# B&R Automation Studio project OpcUaSample410_BrbLibUa103
Automation Studio 4.10.4.38 SP

## Configuration ArSim

CPU PC_any, AutomationRuntime H4.91, Build 6.3.0, Vc V4.16.2

CPU X20CP0483, AutomationRuntime H4.91, Build 6.3.0, Vc V4.16.2

### Task classes (Cpu.sw)
```
Cyclic#1 (cycle 10000 us):
  ClientC <- Tasks.Clients.ClientC.ClientC.prg
  ClientST <- Tasks.Clients.ClientST.ClientST.prg
  SrvMethC <- Tasks.ServerMethods.SrvMethC.SrvMethC.prg
  SrvMethST <- Tasks.ServerMethods.SrvMethST.SrvMethST.prg
  SrvEvntC <- Tasks.ServerEvents.SrvEvntC.SrvEvntC.prg
  SrvEvntST <- Tasks.ServerEvents.SrvEvntST.SrvEvntST.prg [disabled]
  BrbUaCltC <- Tasks.BrbUa.BrbUaClient.BrbUaCltC.BrbUaCltC.prg
  BrbUaCltST <- Tasks.BrbUa.BrbUaClient.BrbUaCltST.BrbUaCltST.prg
  BrbUaSrvC <- Tasks.BrbUa.BrbUaServer.BrbUaSrvC.BrbUaSrvC.prg
  BrbUaSrvST <- Tasks.BrbUa.BrbUaServer.BrbUaSrvST.BrbSrvDatST.prg
  UaCertsC <- Tasks.UaCerts.UaCertsC.UaCertsC.prg
  UaCertsST <- Tasks.UaCerts.UaCertsST.UaCertsST.prg
Cyclic#4 (cycle 100000 us):
  AirCondC <- Tasks.AirCond.AirCondC.AirCondC.prg
  AirCondST <- Tasks.AirCond.AirCondST.AirCondST.prg
Cyclic#7 (cycle 500000 us):
  ServerData <- Tasks.ServerData.ServerData.prg
  SrvDt64C <- Tasks.ServerDt64.SrvDt64C.SrvDt64C.prg
  SrvDt64ST <- Tasks.ServerDt64.ServerDt64ST.SrvDt64ST.prg
  OpcUaAny <- Tasks.OpcUaAny.OpcUaAny.prg
  PubDiag <- Tasks.PubSub.Publisher.PubDiag.prg
  Subscriber <- Tasks.PubSub.Subscriber.Subscriber.prg
  SubDiag <- Tasks.PubSub.Subscriber.SubDiag.prg
Cyclic#8 (cycle 10000 us):
  UtBrbTempl <- UnitTests.UtBrbUaTemplate.prg
  UtBrbUaSta <- UnitTests.UtBrbLibUa.UtBrbUaStatus.prg
  UtBrbUaNod <- UnitTests.UtBrbLibUa.UtBrbUaNodes.prg
  UtBrbUaAtt <- UnitTests.UtBrbLibUa.UtBrbUaAttributes.prg
  UtBrbUaVar <- UnitTests.UtBrbLibUa.UtBrbUaVariantValues.prg
  UtBrbUaByt <- UnitTests.UtBrbLibUa.UtBrbUaByteStrings.prg
  UtBrbUaLoc <- UnitTests.UtBrbLibUa.UtBrbUaLocalizedTexts.prg
  UtBrbUaQua <- UnitTests.UtBrbLibUa.UtBrbUaQualifiedNames.prg
  UtBrbUaTim <- UnitTests.UtBrbLibUa.UtBrbUaTimeAndDate.prg
  UtBrbUaAdd <- UnitTests.UtBrbLibUa.UtBrbUaAdditional.prg
  UtBrbUaCli <- UnitTests.UtBrbLibUa.UtBrbUaClient.prg
  UtBrbUaSer <- UnitTests.UtBrbLibUa.UtBrbUaServer.prg
DataObjects: BrbCltDatC <- Tasks.BrbUa.BrbUaClient.BrbUaCltC.BrbCltDatC.dob, BrbCltDatS <- Tasks.BrbUa.BrbUaClient.BrbUaCltST.BrbCltDatST.dob, BrbSrvDatC <- Tasks.BrbUa.BrbUaServer.BrbUaSrvC.BrbSrvDatC.dob, BrbSrvDatS <- Tasks.BrbUa.BrbUaServer.BrbUaSrvST.BrbSrvDatS.dob
Binaries: TCData, udbdef, TCLang, TC, OpcUaCfg, ashwac, Role, User, ashwd, asfw, arconfig, sysconf, iomap, OpcUa, OpcUaMap
Libraries: UnitTest, UtMgr, UtWs, BrbAsserts, ArCert, ArEventLog, ArPubSubD, ArSsl, AsBrStr, AsBrWStr, AsIecCon, AsOpcUac, AsOpcUas, AsTime, AsUSB, BrbLib, BrbLibUa, Runtime, standard, sys_lib, FileIO, DataObj
```

### Hardware
```
OpcUa_any : OpcUa_any v1.0.0.1  [ETH1 -> PC.IF3 [Cable Type=PowerlinkCable, Length=10, Version=1.0.0.3]]
  ServerDiagnostics = on
  ServerEndpointUrl = opc.tcp://127.0.0.1:4840
  PnPTimeout = 20000
  PnPInitTimeout = 20
  OpcUa_Security_SoftwareCertificates = SslCfgOpcUaClient
  UserIdentifyToken = 1
  Username = Admin
  Password = admin
  Channel1
  ChannelID1 = Read_Usint
  ChannelBrowsePath1 = /0:Root/0:Objects/4:PLC/4:Modules/7:&:&:/7:OpcUaAny/7:Data/7:Read/7:Server/7:nUsint
  ChannelSamplingInterval1 = 500
  ChannelPublishingInterval1 = 500
  ChannelType1 = USINT
  Channel2
  ChannelID2 = Read_Uint
  ChannelBrowsePath2 = /0:Root/0:Objects/4:PLC/4:Modules/7:&:&:/7:OpcUaAny/7:Data/7:Read/7:Server/7:nUint
  ChannelSamplingInterval2 = 500
  ChannelPublishingInterval2 = 500
  ChannelType2 = UINT
  Channel3
  ChannelID3 = Read_Udint
  ChannelBrowsePath3 = /0:Root/0:Objects/4:PLC/4:Modules/7:&:&:/7:OpcUaAny/7:Data/7:Read/7:Server/7:nUdint
  ChannelSamplingInterval3 = 500
  ChannelPublishingInterval3 = 500
  ChannelType3 = UDINT
  Channel4
  ChannelID4 = Write_Usint
  ChannelBrowsePath4 = /0:Root/0:Objects/4:PLC/4:Modules/7:&:&:/7:OpcUaAny/7:Data/7:Write/7:Server/7:nUsint
  ChannelDirection4 = OUT
  ChannelSamplingInterval4 = 500
  ChannelType4 = USINT
  Channel5
  ChannelID5 = Write_Uint
  ChannelBrowsePath5 = /0:Root/0:Objects/4:PLC/4:Modules/7:&:&:/7:OpcUaAny/7:Data/7:Write/7:Server/7:nUint
  ChannelDirection5 = OUT
  ChannelSamplingInterval5 = 500
  ChannelType5 = UINT
  Channel6
  ChannelID6 = Write_Udint
  ChannelBrowsePath6 = /0:Root/0:Objects/4:PLC/4:Modules/7:&:&:/7:OpcUaAny/7:Data/7:Write/7:Server/7:nUdint
  ChannelDirection6 = OUT
  ChannelSamplingInterval6 = 500
  ChannelType6 = UDINT
PC : PC_any v1.1.1.0 (OrderNumber=PC)
  ConfigurationID = OpcUaSample49_ArSim
  Cyclic1Duration = 10000
  Cyclic2Duration = 20000
  Cyclic3Duration = 50000
  Cyclic4Duration = 100000
  Cyclic5Duration = 200000
  Cyclic6Duration = 300000
  Cyclic7Duration = 500000
  Cyclic8Duration = 10000
  ActivateOpcUa = 1
  OpcUaAnonymous = 1
  OpcUaUserName = Admin
  OpcUaPassword = admin  // admin
  OpcUa_Security_AdminRole = Administrators
  OpcUa_Security_SoftwareCertificates = SslCfgOpcUaServer
  OpcUaInformationModels_PV_Version = 2
```

### UaPubSub.uaPubSub - X20CP0483/Connectivity/OpcUA/UaPubSub.uaPubSub
```
Element ExamplePublisher (Type=uaPubSub)
  PublisherId = 3
  NetworkInterface = IF3
  TransportProfileUri = http://opcfoundation.org/UA-Profile/Transport/pubsub-udp-uadp
  Address:
    IpAddress = 239.1.2.3
    Port = 4840
  WriterGroups:
    WriterGroup[1]:
      Name = WriterGroup 500ms
      WriterGroupId = 1
      MaxNetworkMessageSize = 1400
      PublishingInterval = 500
      HeaderLayoutUri = http://opcfoundation.org/UA/PubSub-Layouts/UADP-Periodic-Fixed
      MessageSettingsUadp:
        GroupVersion = 668608188
        DataSetOrdering = 1
      DataSetWriters:
        DataSetWriter[1]:
          Name = DataSetWriter Unsigned
          DataSetWriterId = 1
          PublishedDataSet:
            Name = PublishedDataSet Unsigned
            Publish[1]:
              FieldName = nUsint
              FieldMetaData:
                DataSetFieldId = {ad74a250-bd62-4e87-ba0d-d2bd769ab52c}
                IecTypeCode = 4
                ValueRank = -1
                ArrayDimensions
                IecStringLength = 0
              PublishedPv = ::ServerData:VarsLocal.ReadOnly.nUsint
            Publish[2]:
              FieldName = nUint
              FieldMetaData:
                DataSetFieldId = {f263c076-1c90-4d66-8e4e-e9b1e2cf6b62}
                IecTypeCode = 5
                ValueRank = -1
                ArrayDimensions
                IecStringLength = 0
              PublishedPv = ::ServerData:VarsLocal.ReadOnly.nUint
        DataSetWriter[2]:
          Name = DataSetWriter Signed
          DataSetWriterId = 2
          PublishedDataSet:
            Name = PublishedDataSet Signed
            Publish[1]:
              FieldName = nSint
              FieldMetaData:
                DataSetFieldId = {bcf86e47-32d9-49b1-816e-e7b43017a6e3}
                IecTypeCode = 1
                ValueRank = -1
                ArrayDimensions
                IecStringLength = 0
              PublishedPv = ::ServerData:VarsLocal.ReadOnly.nSint
            Publish[2]:
              FieldName = nInt
              FieldMetaData:
                DataSetFieldId = {3331c223-7101-4ba8-aaad-6da664f841b6}
                IecTypeCode = 2
                ValueRank = -1
                ArrayDimensions
                IecStringLength = 0
              PublishedPv = ::ServerData:VarsLocal.ReadOnly.nInt
    WriterGroup[2]:
      Name = WriterGroup 1000ms
      WriterGroupId = 2
      MaxNetworkMessageSize = 1400
      PublishingInterval = 1000
      HeaderLayoutUri = http://opcfoundation.org/UA/PubSub-Layouts/UADP-Periodic-Fixed
      MessageSettingsUadp:
        GroupVersion = 668611114
        DataSetOrdering = 1
      DataSetWriters:
        DataSetWriter[1]:
          Name = DataSetWriter Array
          DataSetWriterId = 3
          PublishedDataSet:
            Name = PublishedDataSet Array
            Publish[1]:
              FieldName = anInt
              FieldMetaData:
                DataSetFieldId = {ad21bbba-311c-4c33-9ff5-103d2fd11bf2}
                IecTypeCode = 2
                ValueRank = 1
                ArrayDimensions = 5
                IecStringLength = 0
              PublishedPv = ::ServerData:VarsLocal.ReadOnly.anInt
Element ExampleSubscriber (Type=uaPubSub)
  PublisherId = 3
  NetworkInterface = IF3
  TransportProfileUri = http://opcfoundation.org/UA-Profile/Transport/pubsub-udp-uadp
  Address:
    IpAddress = 239.1.2.3
    Port = 4840
  ReaderGroups:
    ReaderGroup[1]:
      Name = ReaderGroup 500ms
      MaxNetworkMessageSize = 1400
      DataSetReaders:
        DataSetReader[1]:
          Name = DataSetReader Unsigned
          PublisherId = 3
          WriterGroupId = 1
          DataSetWriterId = 1
          MessageReceiveTimeout = 2000
          MessageSettingsUadp:
            GroupVersion = 668608188
            NetworkMessageNumber = 1
            DataSetOffset = 15
          TargetVariables:
            Name = ExamplePublisher-WriterGroup 500ms-DataSetWriter Unsigned
            Subscription[1]:
              Source = nUsint
              FieldMetaData:
                DataSetFieldId = {ad74a250-bd62-4e87-ba0d-d2bd769ab52c}
                BuiltInType = 3
                ValueRank = -1
                ArrayDimensions = 
                MaxStringLength = 0
              Target = ::Subscriber:SubscribedData.nUsint
            Subscription[2]:
              Source = nUint
              FieldMetaData:
                DataSetFieldId = {f263c076-1c90-4d66-8e4e-e9b1e2cf6b62}
                BuiltInType = 5
                ValueRank = -1
                ArrayDimensions = 
                MaxStringLength = 0
              Target = ::Subscriber:SubscribedData.nUint
        DataSetReader[2]:
          Name = DataSetReader Signed
          PublisherId = 3
          WriterGroupId = 1
          DataSetWriterId = 2
          MessageReceiveTimeout = 2000
          MessageSettingsUadp:
            GroupVersion = 668608188
            NetworkMessageNumber = 1
            DataSetOffset = 23
          TargetVariables:
            Name = ExamplePublisher-WriterGroup 500ms-DataSetWriter Signed
            Subscription[1]:
              Source = nSint
              FieldMetaData:
                DataSetFieldId = {bcf86e47-32d9-49b1-816e-e7b43017a6e3}
                BuiltInType = 2
                ValueRank = -1
                ArrayDimensions = 
                MaxStringLength = 0
              Target = ::Subscriber:SubscribedData.nSint
            Subscription[2]:
              Source = nInt
              FieldMetaData:
                DataSetFieldId = {3331c223-7101-4ba8-aaad-6da664f841b6}
                BuiltInType = 4
                ValueRank = -1
                ArrayDimensions = 
                MaxStringLength = 0
              Target = ::Subscriber:SubscribedData.nInt
    ReaderGroup[2]:
      Name = ReaderGroup 1000ms
      MaxNetworkMessageSize = 1400
      DataSetReaders:
        DataSetReader[1]:
          Name = DataSetReader Array
          PublisherId = 3
          WriterGroupId = 2
          DataSetWriterId = 3
          MessageReceiveTimeout = 4000
          MessageSettingsUadp:
            GroupVersion = 668611114
            NetworkMessageNumber = 1
            DataSetOffset = 15
          TargetVariables:
            Name = ExamplePublisher-WriterGroup 1000ms-DataSetWriter Array
            Subscription[1]:
              Source = anInt
              FieldMetaData:
                DataSetFieldId = {ad21bbba-311c-4c33-9ff5-103d2fd11bf2}
                BuiltInType = 4
                ValueRank = 1
                ArrayDimensions = 5
                MaxStringLength = 0
              Target = ::Subscriber:SubscribedData.anInt
```

### aircondmodel.uanodeset - X20CP0483/Connectivity/OpcUA/aircondmodel.uanodeset
```
UANodeSet:
  NamespaceUris:
    Uri = http://br-automation.com/AirCondModel/
    Uri = http://opcfoundation.org/UA/DI/
  Models:
    Model (ModelUri=http://br-automation.com/AirCondModel/, PublicationDate=2020-07-13T13:29:09Z, Version=1.0.0)
      RequiredModel (ModelUri=http://opcfoundation.org/UA/, PublicationDate=2018-05-15T00:00:00Z, Version=1.04)
      RequiredModel (ModelUri=http://opcfoundation.org/UA/DI/, PublicationDate=2013-12-02T00:00:00Z, Version=1.01)
  Aliases:
    Alias = i=1 (Alias=Boolean)
    Alias = i=3 (Alias=Byte)
    Alias = i=6 (Alias=Int32)
    Alias = i=10 (Alias=Float)
    Alias = i=12 (Alias=String)
    Alias = i=13 (Alias=DateTime)
    Alias = i=15 (Alias=ByteString)
    Alias = i=21 (Alias=LocalizedText)
    Alias = i=35 (Alias=Organizes)
    Alias = i=37 (Alias=HasModellingRule)
    Alias = i=40 (Alias=HasTypeDefinition)
    Alias = i=41 (Alias=GeneratesEvent)
    Alias = i=45 (Alias=HasSubtype)
    Alias = i=46 (Alias=HasProperty)
    Alias = i=47 (Alias=HasComponent)
    Alias = i=48 (Alias=HasNotifier)
    Alias = i=256 (Alias=IdType)
    Alias = i=291 (Alias=NumericRange)
    Alias = i=296 (Alias=Argument)
    Alias = ns=1;i=3002 (Alias=AirConditionOperationModeType)
  Extensions:
    Extension:
      ModelInfo (Tool=UaModeler, Hash=2Vr1KLh9s9K+CGntyA7k9A==, Version=1.6.2)
  UADataType (NodeId=ns=1;i=3003, BrowseName=1:AirConditionMethodStatusType)
    DisplayName = AirConditionMethodStatusType
    References:
      Reference = i=29 (ReferenceType=HasSubtype, IsForward=false)
      Reference = ns=1;i=6013 (ReferenceType=HasProperty)
    Definition 1:AirConditionMethodStatusType:
      Field Ok = 0
      Field InvalidOperationMode = 1
  UAVariable (DataType=LocalizedText, ParentNodeId=ns=1;i=3003, ValueRank=1, NodeId=ns=1;i=6013, ArrayDimensions=2, BrowseName=EnumStrings)
    DisplayName = EnumStrings
    References:
      Reference = ns=1;i=3003 (ReferenceType=HasProperty, IsForward=false)
      Reference = i=78 (ReferenceType=HasModellingRule)
      Reference = i=68 (ReferenceType=HasTypeDefinition)
    Value:
      ListOfLocalizedText:
        LocalizedText:
          Text = Ok
        LocalizedText:
          Text = InvalidOperationMode
  UADataType (NodeId=ns=1;i=3002, BrowseName=1:AirConditionOperationModeType)
    DisplayName = AirConditionOperationModeType
    Description = Operation mode of an air condition
    References:
      Reference = i=29 (ReferenceType=HasSubtype, IsForward=false)
      Reference = ns=1;i=6008 (ReferenceType=HasProperty)
    Definition 1:AirConditionOperationModeType:
      Field Off = 0
      Field Manual = 1
      Field Automatic = 2
  UAVariable (DataType=LocalizedText, ParentNodeId=ns=1;i=3002, ValueRank=1, NodeId=ns=1;i=6008, ArrayDimensions=3, BrowseName=EnumStrings)
    DisplayName = EnumStrings
    References:
      Reference = ns=1;i=3002 (ReferenceType=HasProperty, IsForward=false)
      Reference = i=78 (ReferenceType=HasModellingRule)
      Reference = i=68 (ReferenceType=HasTypeDefinition)
    Value:
      ListOfLocalizedText:
        LocalizedText:
          Text = Off
        LocalizedText:
          Text = Manual
        LocalizedText:
          Text = Automatic
  UAVariable (SymbolicName=TypeDictionary_BinarySchema, DataType=ByteString, NodeId=ns=1;i=6009, BrowseName=1:TypeDictionary)
    DisplayName = TypeDictionary
    Description = Collects the data type descriptions of http://br-automation.com/AirCondModel/
    References:
      Reference = i=72 (ReferenceType=HasTypeDefinition)
      Reference = ns=1;i=6010 (ReferenceType=HasProperty)
      Reference = i=93 (ReferenceType=HasComponent, IsForward=false)
    Value:
      ByteString = PG9wYzpUeXBlRGljdGlvbmFyeSB4bWxuczp4c2k9Imh0dHA6Ly93d3cudzMub3JnLzIwMDEvWE1MU2NoZ
        W1hLWluc3RhbmNlIiB4bWxuczp0bnM9Imh0dHA6Ly9ici1hdXRvbWF0aW9uLmNvbS9BaXJDb
        25kTW9kZWwvIiBEZWZhdWx0Qnl0ZU9yZGVyPSJMaXR0bGVFbmRpYW4iIHhtbG5zOm9wYz0ia
        HR0cDovL29wY2ZvdW5kYXRpb24ub3JnL0JpbmFyeVNjaGVtYS8iIHhtbG5zOnVhPSJodHRwO
        i8vb3BjZm91bmRhdGlvbi5vcmcvVUEvIiBUYXJnZXROYW1lc3BhY2U9Imh0dHA6Ly9ici1hd
        XRvbWF0aW9uLmNvbS9BaXJDb25kTW9kZWwvIj4KIDxvcGM6SW1wb3J0IE5hbWVzcGFjZT0ia
        HR0cDovL29wY2ZvdW5kYXRpb24ub3JnL1VBLyIvPgogPG9wYzpFbnVtZXJhdGVkVHlwZSBMZ
        W5ndGhJbkJpdHM9IjMyIiBOYW1lPSJBaXJDb25kaXRpb25NZXRob2RTdGF0dXNUeXBlIj4KI
        CA8b3BjOkVudW1lcmF0ZWRWYWx1ZSBOYW1lPSJPayIgVmFsdWU9IjAiLz4KICA8b3BjOkVud
        W1lcmF0ZWRWYWx1ZSBOYW1lPSJJbnZhbGlkT3BlcmF0aW9uTW9kZSIgVmFsdWU9IjEiLz4KI
        Dwvb3BjOkVudW1lcmF0ZWRUeXBlPgogPG9wYzpFbnVtZXJhdGVkVHlwZSBMZW5ndGhJbkJpd
        HM9IjMyIiBOYW1lPSJBaXJDb25kaXRpb25PcGVyYXRpb25Nb2RlVHlwZSI+CiAgPG9wYzpEb
        2N1bWVudGF0aW9uPk9wZXJhdGlvbiBtb2RlIG9mIGFuIGFpciBjb25kaXRpb248L29wYzpEb
        2N1bWVudGF0aW9uPgogIDxvcGM6RW51bWVyYXRlZFZhbHVlIE5hbWU9Ik9mZiIgVmFsdWU9I
        jAiLz4KICA8b3BjOkVudW1lcmF0ZWRWYWx1ZSBOYW1lPSJNYW51YWwiIFZhbHVlPSIxIi8+C
        iAgPG9wYzpFbnVtZXJhdGVkVmFsdWUgTmFtZT0iQXV0b21hdGljIiBWYWx1ZT0iMiIvPgogP
        C9vcGM6RW51bWVyYXRlZFR5cGU+Cjwvb3BjOlR5cGVEaWN0aW9uYXJ5Pgo=
  UAVariable (DataType=String, ParentNodeId=ns=1;i=6009, NodeId=ns=1;i=6010, BrowseName=NamespaceUri)
    DisplayName = NamespaceUri
    References:
      Reference = ns=1;i=6009 (ReferenceType=HasProperty, IsForward=false)
      Reference = i=68 (ReferenceType=HasTypeDefinition)
    Value:
      String = http://br-automation.com/AirCondModel/
  UAVariable (SymbolicName=TypeDictionary_XmlSchema, DataType=ByteString, NodeId=ns=1;i=6011, BrowseName=1:TypeDictionary)
    DisplayName = TypeDictionary
    Description = Collects the data type descriptions of http://br-automation.com/AirCondModel/
    References:
      Reference = i=72 (ReferenceType=HasTypeDefinition)
      Reference = ns=1;i=6012 (ReferenceType=HasProperty)
      Reference = i=92 (ReferenceType=HasComponent, IsForward=false)
    Value:
      ByteString = PHhzOnNjaGVtYSBlbGVtZW50Rm9ybURlZmF1bHQ9InF1YWxpZmllZCIgdGFyZ2V0TmFtZXNwYWNlPSJod
        HRwOi8vYnItYXV0b21hdGlvbi5jb20vQWlyQ29uZE1vZGVsL1R5cGVzLnhzZCIgeG1sbnM6d
        G5zPSJodHRwOi8vYnItYXV0b21hdGlvbi5jb20vQWlyQ29uZE1vZGVsL1R5cGVzLnhzZCIge
        G1sbnM6dWE9Imh0dHA6Ly9vcGNmb3VuZGF0aW9uLm9yZy9VQS8yMDA4LzAyL1R5cGVzLnhzZ
        CIgeG1sbnM6eHM9Imh0dHA6Ly93d3cudzMub3JnLzIwMDEvWE1MU2NoZW1hIj4KIDx4czppb
        XBvcnQgbmFtZXNwYWNlPSJodHRwOi8vb3BjZm91bmRhdGlvbi5vcmcvVUEvMjAwOC8wMi9Ue
        XBlcy54c2QiLz4KIDx4czpzaW1wbGVUeXBlIG5hbWU9IkFpckNvbmRpdGlvbk1ldGhvZFN0Y
        XR1c1R5cGUiPgogIDx4czpyZXN0cmljdGlvbiBiYXNlPSJ4czpzdHJpbmciPgogICA8eHM6Z
        W51bWVyYXRpb24gdmFsdWU9Ik9rXzAiLz4KICAgPHhzOmVudW1lcmF0aW9uIHZhbHVlPSJJb
        nZhbGlkT3BlcmF0aW9uTW9kZV8xIi8+CiAgPC94czpyZXN0cmljdGlvbj4KIDwveHM6c2ltc
        GxlVHlwZT4KIDx4czplbGVtZW50IHR5cGU9InRuczpBaXJDb25kaXRpb25NZXRob2RTdGF0d
        XNUeXBlIiBuYW1lPSJBaXJDb25kaXRpb25NZXRob2RTdGF0dXNUeXBlIi8+CiA8eHM6Y29tc
        GxleFR5cGUgbmFtZT0iTGlzdE9mQWlyQ29uZGl0aW9uTWV0aG9kU3RhdHVzVHlwZSI+CiAgP
        HhzOnNlcXVlbmNlPgogICA8eHM6ZWxlbWVudCBtaW5PY2N1cnM9IjAiIG1heE9jY3Vycz0id
        W5ib3VuZGVkIiB0eXBlPSJ0bnM6QWlyQ29uZGl0aW9uTWV0aG9kU3RhdHVzVHlwZSIgbmFtZ
        T0iQWlyQ29uZGl0aW9uTWV0aG9kU3RhdHVzVHlwZSIgbmlsbGFibGU9InRydWUiLz4KICA8L
        3hzOnNlcXVlbmNlPgogPC94czpjb21wbGV4VHlwZT4KIDx4czplbGVtZW50IHR5cGU9InRuc
        zpMaXN0T2ZBaXJDb25kaXRpb25NZXRob2RTdGF0dXNUeXBlIiBuYW1lPSJMaXN0T2ZBaXJDb
        25kaXRpb25NZXRob2RTdGF0dXNUeXBlIiBuaWxsYWJsZT0idHJ1ZSIvPgogPHhzOnNpbXBsZ
        VR5cGUgbmFtZT0iQWlyQ29uZGl0aW9uT3BlcmF0aW9uTW9kZVR5cGUiPgogIDx4czphbm5vd
        GF0aW9uPgogICA8eHM6ZG9jdW1lbnRhdGlvbj5PcGVyYXRpb24gbW9kZSBvZiBhbiBhaXIgY
        29uZGl0aW9uPC94czpkb2N1bWVudGF0aW9uPgogIDwveHM6YW5ub3RhdGlvbj4KICA8eHM6c
        mVzdHJpY3Rpb24gYmFzZT0ieHM6c3RyaW5nIj4KICAgPHhzOmVudW1lcmF0aW9uIHZhbHVlP
        SJPZmZfMCIvPgogICA8eHM6ZW51bWVyYXRpb24gdmFsdWU9Ik1hbnVhbF8xIi8+CiAgIDx4c
        zplbnVtZXJhdGlvbiB2YWx1ZT0iQXV0b21hdGljXzIiLz4KICA8L3hzOnJlc3RyaWN0aW9uP
        gogPC94czpzaW1wbGVUeXBlPgogPHhzOmVsZW1lbnQgdHlwZT0idG5zOkFpckNvbmRpdGlvb
        k9wZXJhdGlvbk1vZGVUeXBlIiBuYW1lPSJBaXJDb25kaXRpb25PcGVyYXRpb25Nb2RlVHlwZ
        SIvPgogPHhzOmNvbXBsZXhUeXBlIG5hbWU9Ikxpc3RPZkFpckNvbmRpdGlvbk9wZXJhdGlvb
        k1vZGVUeXBlIj4KICA8eHM6c2VxdWVuY2U+CiAgIDx4czplbGVtZW50IG1pbk9jY3Vycz0iM
        CIgbWF4T2NjdXJzPSJ1bmJvdW5kZWQiIHR5cGU9InRuczpBaXJDb25kaXRpb25PcGVyYXRpb
        25Nb2RlVHlwZSIgbmFtZT0iQWlyQ29uZGl0aW9uT3BlcmF0aW9uTW9kZVR5cGUiIG5pbGxhY
        mxlPSJ0cnVlIi8+CiAgPC94czpzZXF1ZW5jZT4KIDwveHM6Y29tcGxleFR5cGU+CiA8eHM6Z
        WxlbWVudCB0eXBlPSJ0bnM6TGlzdE9mQWlyQ29uZGl0aW9uT3BlcmF0aW9uTW9kZVR5cGUiI
        G5hbWU9Ikxpc3RPZkFpckNvbmRpdGlvbk9wZXJhdGlvbk1vZGVUeXBlIiBuaWxsYWJsZT0id
        HJ1ZSIvPgo8L3hzOnNjaGVtYT4K
  UAVariable (DataType=String, ParentNodeId=ns=1;i=6011, NodeId=ns=1;i=6012, BrowseName=NamespaceUri)
    DisplayName = NamespaceUri
    References:
      Reference = ns=1;i=6011 (ReferenceType=HasProperty, IsForward=false)
      Reference = i=68 (ReferenceType=HasTypeDefinition)
    Value:
      String = http://br-automation.com/AirCondModel/Types.xsd
  UAObjectType (NodeId=ns=1;i=1003, BrowseName=1:AirConditionActType)
    DisplayName = AirConditionActType
    Description = Actual values
    References:
      Reference = i=58 (ReferenceType=HasSubtype, IsForward=false)
      Reference = ns=1;i=6016 (ReferenceType=HasComponent)
      Reference = ns=1;i=6017 (ReferenceType=HasComponent)
      Reference = ns=1;i=6018 (ReferenceType=HasComponent)
  UAVariable (DataType=Byte, ParentNodeId=ns=1;i=1003, NodeId=ns=1;i=6016, BrowseName=1:FanLevel)
    DisplayName = FanLevel
    Description = Actual level of the fan
    References:
      Reference = i=63 (ReferenceType=HasTypeDefinition)
      Reference = ns=1;i=1003 (ReferenceType=HasComponent, IsForward=false)
      Reference = i=78 (ReferenceType=HasModellingRule)
  UAVariable (DataType=Int32, ParentNodeId=ns=1;i=1003, NodeId=ns=1;i=6017, BrowseName=1:OperationMode)
    DisplayName = OperationMode
    Description = Actual operation mode of the air condtition: Off, Manual or Auto
    References:
      Reference = i=63 (ReferenceType=HasTypeDefinition)
      Reference = i=78 (ReferenceType=HasModellingRule)
      Reference = ns=1;i=1003 (ReferenceType=HasComponent, IsForward=false)
  UAVariable (DataType=Float, ParentNodeId=ns=1;i=1003, NodeId=ns=1;i=6018, BrowseName=1:Temperature)
    DisplayName = Temperature
    Description = Actual room temperature
    References:
      Reference = i=63 (ReferenceType=HasTypeDefinition)
      Reference = i=78 (ReferenceType=HasModellingRule)
      Reference = ns=1;i=1003 (ReferenceType=HasComponent, IsForward=false)
  UAObjectType (NodeId=ns=1;i=1004, BrowseName=1:AirConditionSetType)
    DisplayName = AirConditionSetType
    Description = Set values
    References:
      Reference = i=58 (ReferenceType=HasSubtype, IsForward=false)
      Reference = ns=1;i=6019 (ReferenceType=HasComponent)
      Reference = ns=1;i=6020 (ReferenceType=HasComponent)
  UAVariable (DataType=Byte, ParentNodeId=ns=1;i=1004, NodeId=ns=1;i=6019, BrowseName=1:FanLevel, AccessLevel=3)
    DisplayName = FanLevel
    Description = The set fan level for operation mode manual
    References:
      Reference = i=63 (ReferenceType=HasTypeDefinition)
      Reference = ns=1;i=1004 (ReferenceType=HasComponent, IsForward=false)
      Reference = i=78 (ReferenceType=HasModellingRule)
  UAVariable (DataType=Float, ParentNodeId=ns=1;i=1004, NodeId=ns=1;i=6020, BrowseName=1:Temperature, AccessLevel=3)
    DisplayName = Temperature
    Description = The set temperature for operation mode automatic
    References:
      Reference = i=63 (ReferenceType=HasTypeDefinition)
      Reference = i=78 (ReferenceType=HasModellingRule)
      Reference = ns=1;i=1004 (ReferenceType=HasComponent, IsForward=false)
  UAObjectType (NodeId=ns=1;i=1006, BrowseName=1:AirConditionsType)
    DisplayName = AirConditionsType
    Description = Air conditions
    References:
      Reference = i=58 (ReferenceType=HasSubtype, IsForward=false)
      Reference = ns=1;i=5004 (ReferenceType=HasComponent)
      Reference = ns=1;i=5007 (ReferenceType=HasComponent)
      Reference = ns=1;i=5010 (ReferenceType=HasComponent)
  UAObject (ParentNodeId=ns=1;i=1006, NodeId=ns=1;i=5004, BrowseName=1:BedRoom)
    DisplayName = BedRoom
    Description = Bed room air condition
    References:
      Reference = ns=1;i=5005 (ReferenceType=HasComponent)
      Reference = ns=1;i=1005 (ReferenceType=HasTypeDefinition)
      Reference = ns=1;i=1006 (ReferenceType=HasComponent, IsForward=false)
      Reference = i=78 (ReferenceType=HasModellingRule)
      Reference = ns=1;i=6092 (ReferenceType=HasComponent)
      Reference = ns=1;i=5006 (ReferenceType=HasComponent)
      Reference = ns=1;i=7002 (ReferenceType=HasComponent)
  UAObject (ParentNodeId=ns=1;i=5004, NodeId=ns=1;i=5005, BrowseName=1:Act)
    DisplayName = Act
    Description = Actual values
    References:
      Reference = ns=1;i=5004 (ReferenceType=HasComponent, IsForward=false)
      Reference = ns=1;i=1003 (ReferenceType=HasTypeDefinition)
      Reference = ns=1;i=6026 (ReferenceType=HasComponent)
      Reference = i=78 (ReferenceType=HasModellingRule)
      Reference = ns=1;i=6027 (ReferenceType=HasComponent)
      Reference = ns=1;i=6028 (ReferenceType=HasComponent)
  UAVariable (DataType=Byte, ParentNodeId=ns=1;i=5005, NodeId=ns=1;i=6026, BrowseName=1:FanLevel)
    DisplayName = FanLevel
    Description = Actual level of the fan
    References:
      Reference = i=63 (ReferenceType=HasTypeDefinition)
      Reference = ns=1;i=5005 (ReferenceType=HasComponent, IsForward=false)
      Reference = i=78 (ReferenceType=HasModellingRule)
  UAVariable (DataType=Int32, ParentNodeId=ns=1;i=5005, NodeId=ns=1;i=6027, BrowseName=1:OperationMode)
    DisplayName = OperationMode
    Description = Actual operation mode of the air condtition: Off, Manual or Auto
    References:
      Reference = i=63 (ReferenceType=HasTypeDefinition)
      Reference = i=78 (ReferenceType=HasModellingRule)
      Reference = ns=1;i=5005 (ReferenceType=HasComponent, IsForward=false)
  UAVariable (DataType=Float, ParentNodeId=ns=1;i=5005, NodeId=ns=1;i=6028, BrowseName=1:Temperature)
    DisplayName = Temperature
    Description = Actual room temperature
    References:
      Reference = i=63 (ReferenceType=HasTypeDefinition)
      Reference = i=78 (ReferenceType=HasModellingRule)
      Reference = ns=1;i=5005 (ReferenceType=HasComponent, IsForward=false)
  UAVariable (DataType=String, ParentNodeId=ns=1;i=5004, NodeId=ns=1;i=6092, BrowseName=1:Name)
    DisplayName = Name
    Description = Name of the instance
    References:
      Reference = i=63 (ReferenceType=HasTypeDefinition)
      Reference = i=78 (ReferenceType=HasModellingRule)
      Reference = ns=1;i=5004 (ReferenceType=HasComponent, IsForward=false)
  UAObject (ParentNodeId=ns=1;i=5004, NodeId=ns=1;i=5006, BrowseName=1:Set)
    DisplayName = Set
    Description = Set values
    References:
      Reference = ns=1;i=1004 (ReferenceType=HasTypeDefinition)
      Reference = ns=1;i=6029 (ReferenceType=HasComponent)
      Reference = i=78 (ReferenceType=HasModellingRule)
      Reference = ns=1;i=5004 (ReferenceType=HasComponent, IsForward=false)
      Reference = ns=1;i=6030 (ReferenceType=HasComponent)
  UAVariable (DataType=Byte, ParentNodeId=ns=1;i=5006, NodeId=ns=1;i=6029, BrowseName=1:FanLevel, AccessLevel=3)
    DisplayName = FanLevel
    Description = The set fan level for operation mode manual
    References:
      Reference = i=63 (ReferenceType=HasTypeDefinition)
      Reference = ns=1;i=5006 (ReferenceType=HasComponent, IsForward=false)
      Reference = i=78 (ReferenceType=HasModellingRule)
  UAVariable (DataType=Float, ParentNodeId=ns=1;i=5006, NodeId=ns=1;i=6030, BrowseName=1:Temperature, AccessLevel=3)
    DisplayName = Temperature
    Description = The set temperature for operation mode automatic
    References:
      Reference = i=63 (ReferenceType=HasTypeDefinition)
      Reference = i=78 (ReferenceType=HasModellingRule)
      Reference = ns=1;i=5006 (ReferenceType=HasComponent, IsForward=false)
  UAMethod (ParentNodeId=ns=1;i=5004, NodeId=ns=1;i=7002, BrowseName=1:SetOperationMode, MethodDeclarationId=ns=1;i=7001)
    DisplayName = SetOperationMode
    Description = Set the operation mode of the air condition to Off, Manual or Auto
    References:
      Reference = ns=1;i=6057 (ReferenceType=HasProperty)
      Reference = i=78 (ReferenceType=HasModellingRule)
      Reference = ns=1;i=6064 (ReferenceType=HasProperty)
      Reference = ns=1;i=5004 (ReferenceType=HasComponent, IsForward=false)
  UAVariable (DataType=Argument, ParentNodeId=ns=1;i=7002, ValueRank=1, NodeId=ns=1;i=6057, ArrayDimensions=1, BrowseName=InputArguments)
    DisplayName = InputArguments
    References:
      Reference = i=78 (ReferenceType=HasModellingRule)
      Reference = i=68 (ReferenceType=HasTypeDefinition)
      Reference = ns=1;i=7002 (ReferenceType=HasProperty, IsForward=false)
    Value:
      ListOfExtensionObject:
        ExtensionObject:
          TypeId:
            Identifier = i=297
          Body:
            Argument:
              Name = OperationMode
              DataType:
                Identifier = ns=1;i=3002
              ValueRank = -1
              ArrayDimensions
              Description:
                Text = OperationMode (Off, Manual or Automatic)
  UAVariable (DataType=Argument, ParentNodeId=ns=1;i=7002, ValueRank=1, NodeId=ns=1;i=6064, ArrayDimensions=1, BrowseName=OutputArguments)
    DisplayName = OutputArguments
    References:
      Reference = i=78 (ReferenceType=HasModellingRule)
      Reference = i=68 (ReferenceType=HasTypeDefinition)
      Reference = ns=1;i=7002 (ReferenceType=HasProperty, IsForward=false)
    Value:
      ListOfExtensionObject:
        ExtensionObject:
          TypeId:
            Identifier = i=297
          Body:
            Argument:
              Name = Status
              DataType:
                Identifier = ns=1;i=3003
              ValueRank = -1
              ArrayDimensions
              Description:
                Text = Status of the method
  UAObject (ParentNodeId=ns=1;i=1006, NodeId=ns=1;i=5007, BrowseName=1:Corridor)
    DisplayName = Corridor
    Description = Corridor air condition
    References:
      Reference = ns=1;i=5008 (ReferenceType=HasComponent)
      Reference = ns=1;i=1005 (ReferenceType=HasTypeDefinition)
      Reference = ns=1;i=1006 (ReferenceType=HasComponent, IsForward=false)
      Reference = i=78 (ReferenceType=HasModellingRule)
      Reference = ns=1;i=6093 (ReferenceType=HasComponent)
      Reference = ns=1;i=5009 (ReferenceType=HasComponent)
      Reference = ns=1;i=7003 (ReferenceType=HasComponent)
  UAObject (ParentNodeId=ns=1;i=5007, NodeId=ns=1;i=5008, BrowseName=1:Act)
    DisplayName = Act
    Description = Actual values
    References:
      Reference = ns=1;i=5007 (ReferenceType=HasComponent, IsForward=false)
      Reference = ns=1;i=1003 (ReferenceType=HasTypeDefinition)
      Reference = ns=1;i=6031 (ReferenceType=HasComponent)
      Reference = i=78 (ReferenceType=HasModellingRule)
      Reference = ns=1;i=6032 (ReferenceType=HasComponent)
      Reference = ns=1;i=6033 (ReferenceType=HasComponent)
  UAVariable (DataType=Byte, ParentNodeId=ns=1;i=5008, NodeId=ns=1;i=6031, BrowseName=1:FanLevel)
    DisplayName = FanLevel
    Description = Actual level of the fan
    References:
      Reference = i=63 (ReferenceType=HasTypeDefinition)
      Reference = ns=1;i=5008 (ReferenceType=HasComponent, IsForward=false)
      Reference = i=78 (ReferenceType=HasModellingRule)
  UAVariable (DataType=Int32, ParentNodeId=ns=1;i=5008, NodeId=ns=1;i=6032, BrowseName=1:OperationMode)
    DisplayName = OperationMode
    Description = Actual operation mode of the air condtition: Off, Manual or Auto
    References:
      Reference = i=63 (ReferenceType=HasTypeDefinition)
      Reference = i=78 (ReferenceType=HasModellingRule)
      Reference = ns=1;i=5008 (ReferenceType=HasComponent, IsForward=false)
  UAVariable (DataType=Float, ParentNodeId=ns=1;i=5008, NodeId=ns=1;i=6033, BrowseName=1:Temperature)
    DisplayName = Temperature
    Description = Actual room temperature
    References:
      Reference = i=63 (ReferenceType=HasTypeDefinition)
      Reference = i=78 (ReferenceType=HasModellingRule)
      Reference = ns=1;i=5008 (ReferenceType=HasComponent, IsForward=false)
  UAVariable (DataType=String, ParentNodeId=ns=1;i=5007, NodeId=ns=1;i=6093, BrowseName=1:Name)
    DisplayName = Name
    Description = Name of the instance
    References:
      Reference = i=63 (ReferenceType=HasTypeDefinition)
      Reference = i=78 (ReferenceType=HasModellingRule)
      Reference = ns=1;i=5007 (ReferenceType=HasComponent, IsForward=false)
  UAObject (ParentNodeId=ns=1;i=5007, NodeId=ns=1;i=5009, BrowseName=1:Set)
    DisplayName = Set
    Description = Set values
    References:
      Reference = ns=1;i=1004 (ReferenceType=HasTypeDefinition)
      Reference = ns=1;i=6034 (ReferenceType=HasComponent)
      Reference = i=78 (ReferenceType=HasModellingRule)
      Reference = ns=1;i=5007 (ReferenceType=HasComponent, IsForward=false)
      Reference = ns=1;i=6035 (ReferenceType=HasComponent)
  UAVariable (DataType=Byte, ParentNodeId=ns=1;i=5009, NodeId=ns=1;i=6034, BrowseName=1:FanLevel, AccessLevel=3)
    DisplayName = FanLevel
    Description = The set fan level for operation mode manual
    References:
      Reference = i=63 (ReferenceType=HasTypeDefinition)
      Reference = ns=1;i=5009 (ReferenceType=HasComponent, IsForward=false)
      Reference = i=78 (ReferenceType=HasModellingRule)
  UAVariable (DataType=Float, ParentNodeId=ns=1;i=5009, NodeId=ns=1;i=6035, BrowseName=1:Temperature, AccessLevel=3)
    DisplayName = Temperature
    Description = The set temperature for operation mode automatic
    References:
      Reference = i=63 (ReferenceType=HasTypeDefinition)
      Reference = i=78 (ReferenceType=HasModellingRule)
      Reference = ns=1;i=5009 (ReferenceType=HasComponent, IsForward=false)
  UAMethod (ParentNodeId=ns=1;i=5007, NodeId=ns=1;i=7003, BrowseName=1:SetOperationMode, MethodDeclarationId=ns=1;i=7001)
    DisplayName = SetOperationMode
    Description = Set the operation mode of the air condition to Off, Manual or Auto
    References:
      Reference = ns=1;i=6058 (ReferenceType=HasProperty)
      Reference = i=78 (ReferenceType=HasModellingRule)
      Reference = ns=1;i=6065 (ReferenceType=HasProperty)
      Reference = ns=1;i=5007 (ReferenceType=HasComponent, IsForward=false)
  UAVariable (DataType=Argument, ParentNodeId=ns=1;i=7003, ValueRank=1, NodeId=ns=1;i=6058, ArrayDimensions=1, BrowseName=InputArguments)
    DisplayName = InputArguments
    References:
      Reference = i=78 (ReferenceType=HasModellingRule)
      Reference = i=68 (ReferenceType=HasTypeDefinition)
      Reference = ns=1;i=7003 (ReferenceType=HasProperty, IsForward=false)
    Value:
      ListOfExtensionObject:
        ExtensionObject:
          TypeId:
            Identifier = i=297
          Body:
            Argument:
              Name = OperationMode
              DataType:
                Identifier = ns=1;i=3002
              ValueRank = -1
              ArrayDimensions
              Description:
                Text = OperationMode (Off, Manual or Automatic)
  UAVariable (DataType=Argument, ParentNodeId=ns=1;i=7003, ValueRank=1, NodeId=ns=1;i=6065, ArrayDimensions=1, BrowseName=OutputArguments)
    DisplayName = OutputArguments
    References:
      Reference = i=78 (ReferenceType=HasModellingRule)
      Reference = i=68 (ReferenceType=HasTypeDefinition)
      Reference = ns=1;i=7003 (ReferenceType=HasProperty, IsForward=false)
    Value:
      ListOfExtensionObject:
        ExtensionObject:
          TypeId:
            Identifier = i=297
          Body:
            Argument:
              Name = Status
              DataType:
                Identifier = ns=1;i=3003
              ValueRank = -1
              ArrayDimensions
              Description:
                Text = Status of the method
  UAObject (ParentNodeId=ns=1;i=1006, NodeId=ns=1;i=5010, BrowseName=1:LivingRoom)
    DisplayName = LivingRoom
    Description = Living room air condition
    References:
      Reference = ns=1;i=5011 (ReferenceType=HasComponent)
      Reference = ns=1;i=1005 (ReferenceType=HasTypeDefinition)
      Reference = ns=1;i=1006 (ReferenceType=HasComponent, IsForward=false)
      Reference = i=78 (ReferenceType=HasModellingRule)
      Reference = ns=1;i=6094 (ReferenceType=HasComponent)
      Reference = ns=1;i=5012 (ReferenceType=HasComponent)
      Reference = ns=1;i=7004 (ReferenceType=HasComponent)
  UAObject (ParentNodeId=ns=1;i=5010, NodeId=ns=1;i=5011, BrowseName=1:Act)
    DisplayName = Act
    Description = Actual values
    References:
      Reference = ns=1;i=5010 (ReferenceType=HasComponent, IsForward=false)
      Reference = ns=1;i=1003 (ReferenceType=HasTypeDefinition)
      Reference = ns=1;i=6036 (ReferenceType=HasComponent)
      Reference = i=78 (ReferenceType=HasModellingRule)
      Reference = ns=1;i=6037 (ReferenceType=HasComponent)
      Reference = ns=1;i=6038 (ReferenceType=HasComponent)
  UAVariable (DataType=Byte, ParentNodeId=ns=1;i=5011, NodeId=ns=1;i=6036, BrowseName=1:FanLevel)
    DisplayName = FanLevel
    Description = Actual level of the fan
    References:
      Reference = i=63 (ReferenceType=HasTypeDefinition)
      Reference = ns=1;i=5011 (ReferenceType=HasComponent, IsForward=false)
      Reference = i=78 (ReferenceType=HasModellingRule)
  UAVariable (DataType=Int32, ParentNodeId=ns=1;i=5011, NodeId=ns=1;i=6037, BrowseName=1:OperationMode)
    DisplayName = OperationMode
    Description = Actual operation mode of the air condtition: Off, Manual or Auto
    References:
      Reference = i=63 (ReferenceType=HasTypeDefinition)
      Reference = i=78 (ReferenceType=HasModellingRule)
      Reference = ns=1;i=5011 (ReferenceType=HasComponent, IsForward=false)
  UAVariable (DataType=Float, ParentNodeId=ns=1;i=5011, NodeId=ns=1;i=6038, BrowseName=1:Temperature)
    DisplayName = Temperature
    Description = Actual room temperature
    References:
      Reference = i=63 (ReferenceType=HasTypeDefinition)
      Reference = i=78 (ReferenceType=HasModellingRule)
      Reference = ns=1;i=5011 (ReferenceType=HasComponent, IsForward=false)
  UAVariable (DataType=String, ParentNodeId=ns=1;i=5010, NodeId=ns=1;i=6094, BrowseName=1:Name)
    DisplayName = Name
    Description = Name of the instance
    References:
      Reference = i=63 (ReferenceType=HasTypeDefinition)
      Reference = i=78 (ReferenceType=HasModellingRule)
      Reference = ns=1;i=5010 (ReferenceType=HasComponent, IsForward=false)
  UAObject (ParentNodeId=ns=1;i=5010, NodeId=ns=1;i=5012, BrowseName=1:Set)
    DisplayName = Set
    Description = Set values
    References:
      Reference = ns=1;i=1004 (ReferenceType=HasTypeDefinition)
      Reference = ns=1;i=6039 (ReferenceType=HasComponent)
      Reference = i=78 (ReferenceType=HasModellingRule)
      Reference = ns=1;i=5010 (ReferenceType=HasComponent, IsForward=false)
      Reference = ns=1;i=6040 (ReferenceType=HasComponent)
  UAVariable (DataType=Byte, ParentNodeId=ns=1;i=5012, NodeId=ns=1;i=6039, BrowseName=1:FanLevel, AccessLevel=3)
    DisplayName = FanLevel
    Description = The set fan level for operation mode manual
    References:
      Reference = i=63 (ReferenceType=HasTypeDefinition)
      Reference = ns=1;i=5012 (ReferenceType=HasComponent, IsForward=false)
      Reference = i=78 (ReferenceType=HasModellingRule)
  UAVariable (DataType=Float, ParentNodeId=ns=1;i=5012, NodeId=ns=1;i=6040, BrowseName=1:Temperature, AccessLevel=3)
    DisplayName = Temperature
    Description = The set temperature for operation mode automatic
    References:
      Reference = i=63 (ReferenceType=HasTypeDefinition)
      Reference = i=78 (ReferenceType=HasModellingRule)
      Reference = ns=1;i=5012 (ReferenceType=HasComponent, IsForward=false)
  UAMethod (ParentNodeId=ns=1;i=5010, NodeId=ns=1;i=7004, BrowseName=1:SetOperationMode, MethodDeclarationId=ns=1;i=7001)
    DisplayName = SetOperationMode
    Description = Set the operation mode of the air condition to Off, Manual or Auto
    References:
      Reference = ns=1;i=6059 (ReferenceType=HasProperty)
      Reference = i=78 (ReferenceType=HasModellingRule)
      Reference = ns=1;i=6066 (ReferenceType=HasProperty)
      Reference = ns=1;i=5010 (ReferenceType=HasComponent, IsForward=false)
  UAVariable (DataType=Argument, ParentNodeId=ns=1;i=7004, ValueRank=1, NodeId=ns=1;i=6059, ArrayDimensions=1, BrowseName=InputArguments)
    DisplayName = InputArguments
    References:
      Reference = i=78 (ReferenceType=HasModellingRule)
      Reference = i=68 (ReferenceType=HasTypeDefinition)
      Reference = ns=1;i=7004 (ReferenceType=HasProperty, IsForward=false)
    Value:
      ListOfExtensionObject:
        ExtensionObject:
          TypeId:
            Identifier = i=297
          Body:
            Argument:
              Name = OperationMode
              DataType:
                Identifier = ns=1;i=3002
              ValueRank = -1
              ArrayDimensions
              Description:
                Text = OperationMode (Off, Manual or Automatic)
  UAVariable (DataType=Argument, ParentNodeId=ns=1;i=7004, ValueRank=1, NodeId=ns=1;i=6066, ArrayDimensions=1, BrowseName=OutputArguments)
    DisplayName = OutputArguments
    References:
      Reference = i=78 (ReferenceType=HasModellingRule)
      Reference = i=68 (ReferenceType=HasTypeDefinition)
      Reference = ns=1;i=7004 (ReferenceType=HasProperty, IsForward=false)
    Value:
      ListOfExtensionObject:
        ExtensionObject:
          TypeId:
            Identifier = i=297
          Body:
            Argument:
              Name = Status
              DataType:
                Identifier = ns=1;i=3003
              ValueRank = -1
              ArrayDimensions
              Description:
                Text = Status of the method
  UAObjectType (NodeId=ns=1;i=1005, BrowseName=1:AirConditionType)
    DisplayName = AirConditionType
    Description = Air condition
    References:
      Reference = ns=1;i=5002 (ReferenceType=HasComponent)
      Reference = ns=1;i=1002 (ReferenceType=GeneratesEvent)
      Reference = i=58 (ReferenceType=HasSubtype, IsForward=false)
      Reference = ns=1;i=6091 (ReferenceType=HasComponent)
      Reference = ns=1;i=5003 (ReferenceType=HasComponent)
      Reference = ns=1;i=7001 (ReferenceType=HasComponent)
  UAObject (ParentNodeId=ns=1;i=1005, NodeId=ns=1;i=5002, BrowseName=1:Act)
    DisplayName = Act
    Description = Actual values
    References:
      Reference = ns=1;i=1005 (ReferenceType=HasComponent, IsForward=false)
      Reference = ns=1;i=1003 (ReferenceType=HasTypeDefinition)
      Reference = ns=1;i=6021 (ReferenceType=HasComponent)
      Reference = i=78 (ReferenceType=HasModellingRule)
      Reference = ns=1;i=6022 (ReferenceType=HasComponent)
      Reference = ns=1;i=6023 (ReferenceType=HasComponent)
  UAVariable (DataType=Byte, ParentNodeId=ns=1;i=5002, NodeId=ns=1;i=6021, BrowseName=1:FanLevel)
    DisplayName = FanLevel
    Description = Actual level of the fan
    References:
      Reference = i=63 (ReferenceType=HasTypeDefinition)
      Reference = ns=1;i=5002 (ReferenceType=HasComponent, IsForward=false)
      Reference = i=78 (ReferenceType=HasModellingRule)
  UAVariable (DataType=Int32, ParentNodeId=ns=1;i=5002, NodeId=ns=1;i=6022, BrowseName=1:OperationMode)
    DisplayName = OperationMode
    Description = Actual operation mode of the air condtition: Off, Manual or Auto
    References:
      Reference = i=63 (ReferenceType=HasTypeDefinition)
      Reference = i=78 (ReferenceType=HasModellingRule)
      Reference = ns=1;i=5002 (ReferenceType=HasComponent, IsForward=false)
  UAVariable (DataType=Float, ParentNodeId=ns=1;i=5002, NodeId=ns=1;i=6023, BrowseName=1:Temperature)
    DisplayName = Temperature
    Description = Actual room temperature
    References:
      Reference = i=63 (ReferenceType=HasTypeDefinition)
      Reference = i=78 (ReferenceType=HasModellingRule)
      Reference = ns=1;i=5002 (ReferenceType=HasComponent, IsForward=false)
  UAVariable (DataType=String, ParentNodeId=ns=1;i=1005, NodeId=ns=1;i=6091, BrowseName=1:Name)
    DisplayName = Name
    Description = Name of the instance
    References:
      Reference = i=63 (ReferenceType=HasTypeDefinition)
      Reference = i=78 (ReferenceType=HasModellingRule)
      Reference = ns=1;i=1005 (ReferenceType=HasComponent, IsForward=false)
  UAObject (ParentNodeId=ns=1;i=1005, NodeId=ns=1;i=5003, BrowseName=1:Set)
    DisplayName = Set
    Description = Set values
    References:
      Reference = ns=1;i=1004 (ReferenceType=HasTypeDefinition)
      Reference = ns=1;i=6024 (ReferenceType=HasComponent)
      Reference = i=78 (ReferenceType=HasModellingRule)
      Reference = ns=1;i=1005 (ReferenceType=HasComponent, IsForward=false)
      Reference = ns=1;i=6025 (ReferenceType=HasComponent)
  UAVariable (DataType=Byte, ParentNodeId=ns=1;i=5003, NodeId=ns=1;i=6024, BrowseName=1:FanLevel, AccessLevel=3)
    DisplayName = FanLevel
    Description = The set fan level for operation mode manual
    References:
      Reference = i=63 (ReferenceType=HasTypeDefinition)
      Reference = ns=1;i=5003 (ReferenceType=HasComponent, IsForward=false)
      Reference = i=78 (ReferenceType=HasModellingRule)
  UAVariable (DataType=Float, ParentNodeId=ns=1;i=5003, NodeId=ns=1;i=6025, BrowseName=1:Temperature, AccessLevel=3)
    DisplayName = Temperature
    Description = The set temperature for operation mode automatic
    References:
      Reference = i=63 (ReferenceType=HasTypeDefinition)
      Reference = i=78 (ReferenceType=HasModellingRule)
      Reference = ns=1;i=5003 (ReferenceType=HasComponent, IsForward=false)
  UAMethod (ParentNodeId=ns=1;i=1005, NodeId=ns=1;i=7001, BrowseName=1:SetOperationMode)
    DisplayName = SetOperationMode
    Description = Set the operation mode of the air condition to Off, Manual or Auto
    References:
      Reference = ns=1;i=6056 (ReferenceType=HasProperty)
      Reference = i=78 (ReferenceType=HasModellingRule)
      Reference = ns=1;i=6063 (ReferenceType=HasProperty)
      Reference = ns=1;i=1005 (ReferenceType=HasComponent, IsForward=false)
  UAVariable (DataType=Argument, ParentNodeId=ns=1;i=7001, ValueRank=1, NodeId=ns=1;i=6056, ArrayDimensions=1, BrowseName=InputArguments)
    DisplayName = InputArguments
    References:
      Reference = i=78 (ReferenceType=HasModellingRule)
      Reference = i=68 (ReferenceType=HasTypeDefinition)
      Reference = ns=1;i=7001 (ReferenceType=HasProperty, IsForward=false)
    Value:
      ListOfExtensionObject:
        ExtensionObject:
          TypeId:
            Identifier = i=297
          Body:
            Argument:
              Name = OperationMode
              DataType:
                Identifier = ns=1;i=3002
              ValueRank = -1
              ArrayDimensions
              Description:
                Text = OperationMode (Off, Manual or Automatic)
  UAVariable (DataType=Argument, ParentNodeId=ns=1;i=7001, ValueRank=1, NodeId=ns=1;i=6063, ArrayDimensions=1, BrowseName=OutputArguments)
    DisplayName = OutputArguments
    References:
      Reference = i=78 (ReferenceType=HasModellingRule)
      Reference = i=68 (ReferenceType=HasTypeDefinition)
      Reference = ns=1;i=7001 (ReferenceType=HasProperty, IsForward=false)
    Value:
      ListOfExtensionObject:
        ExtensionObject:
          TypeId:
            Identifier = i=297
          Body:
            Argument:
              Name = Status
              DataType:
                Identifier = ns=1;i=3003
              ValueRank = -1
              ArrayDimensions
              Description:
                Text = Status of the method
  UAObjectType (NodeId=ns=1;i=1002, BrowseName=1:AirConditionOperationModeChanged)
    DisplayName = AirConditionOperationModeChanged
    References:
      Reference = i=2041 (ReferenceType=HasSubtype, IsForward=false)
      Reference = ns=1;i=6015 (ReferenceType=HasProperty)
      Reference = ns=1;i=6014 (ReferenceType=HasProperty)
      Reference = ns=1;i=1005 (ReferenceType=GeneratesEvent, IsForward=false)
      Reference = ns=1;i=5013 (ReferenceType=GeneratesEvent, IsForward=false)
      Reference = ns=1;i=5017 (ReferenceType=GeneratesEvent, IsForward=false)
      Reference = ns=1;i=5020 (ReferenceType=GeneratesEvent, IsForward=false)
      Reference = ns=1;i=5023 (ReferenceType=GeneratesEvent, IsForward=false)
      Reference = ns=1;i=5027 (ReferenceType=GeneratesEvent, IsForward=false)
      Reference = ns=1;i=5030 (ReferenceType=GeneratesEvent, IsForward=false)
      Reference = ns=1;i=5033 (ReferenceType=GeneratesEvent, IsForward=false)
  UAVariable (DataType=AirConditionOperationModeType, ParentNodeId=ns=1;i=1002, NodeId=ns=1;i=6015, BrowseName=1:NewOperationMode)
    DisplayName = NewOperationMode
    Description = Operation mode after change
    References:
      Reference = i=78 (ReferenceType=HasModellingRule)
      Reference = ns=1;i=1002 (ReferenceType=HasProperty, IsForward=false)
      Reference = i=68 (ReferenceType=HasTypeDefinition)
  UAVariable (DataType=AirConditionOperationModeType, ParentNodeId=ns=1;i=1002, NodeId=ns=1;i=6014, BrowseName=1:OldOperationMode)
    DisplayName = OldOperationMode
    Description = Operation mode before change
    References:
      Reference = i=78 (ReferenceType=HasModellingRule)
      Reference = ns=1;i=1002 (ReferenceType=HasProperty, IsForward=false)
      Reference = i=68 (ReferenceType=HasTypeDefinition)
  UAObject (NodeId=ns=1;i=5033, BrowseName=1:AirConditions)
    DisplayName = AirConditions
    Description = Root of all air conditions in variants of ANSI-C and StructuredText
    References:
      Reference = ns=1;i=1002 (ReferenceType=GeneratesEvent)
      Reference = ns=2;i=5001 (ReferenceType=Organizes, IsForward=false)
      Reference = i=58 (ReferenceType=HasTypeDefinition)
      Reference = ns=1;i=5014 (ReferenceType=Organizes)
      Reference = ns=1;i=5024 (ReferenceType=Organizes)
  UAObject (NodeId=ns=1;i=5014, BrowseName=1:C)
    DisplayName = C
    Description = Root of all air conditions in variant of ANSI-C
    References:
      Reference = ns=1;i=1006 (ReferenceType=HasTypeDefinition)
      Reference = ns=1;i=5013 (ReferenceType=HasComponent)
      Reference = ns=1;i=5017 (ReferenceType=HasComponent)
      Reference = ns=1;i=5020 (ReferenceType=HasComponent)
      Reference = ns=1;i=5033 (ReferenceType=Organizes, IsForward=false)
  UAObject (ParentNodeId=ns=1;i=5014, EventNotifier=1, NodeId=ns=1;i=5013, BrowseName=1:BedRoom)
    DisplayName = BedRoom
    Description = Bed room air condition
    References:
      Reference = ns=1;i=5015 (ReferenceType=HasComponent)
      Reference = ns=1;i=1002 (ReferenceType=GeneratesEvent)
      Reference = ns=1;i=1005 (ReferenceType=HasTypeDefinition)
      Reference = ns=1;i=6095 (ReferenceType=HasComponent)
      Reference = ns=1;i=5016 (ReferenceType=HasComponent)
      Reference = ns=1;i=7005 (ReferenceType=HasComponent)
      Reference = i=2253 (ReferenceType=HasNotifier, IsForward=false)
      Reference = ns=1;i=5014 (ReferenceType=HasComponent, IsForward=false)
  UAObject (ParentNodeId=ns=1;i=5013, NodeId=ns=1;i=5015, BrowseName=1:Act)
    DisplayName = Act
    Description = Actual values
    References:
      Reference = ns=1;i=5013 (ReferenceType=HasComponent, IsForward=false)
      Reference = ns=1;i=1003 (ReferenceType=HasTypeDefinition)
      Reference = ns=1;i=6041 (ReferenceType=HasComponent)
      Reference = ns=1;i=6042 (ReferenceType=HasComponent)
      Reference = ns=1;i=6043 (ReferenceType=HasComponent)
  UAVariable (DataType=Byte, ParentNodeId=ns=1;i=5015, NodeId=ns=1;i=6041, BrowseName=1:FanLevel)
    DisplayName = FanLevel
    Description = Actual level of the fan
    References:
      Reference = i=63 (ReferenceType=HasTypeDefinition)
      Reference = ns=1;i=5015 (ReferenceType=HasComponent, IsForward=false)
  UAVariable (DataType=Int32, ParentNodeId=ns=1;i=5015, NodeId=ns=1;i=6042, BrowseName=1:OperationMode)
    DisplayName = OperationMode
    Description = Actual operation mode of the air condtition: Off, Manual or Auto
    References:
      Reference = i=63 (ReferenceType=HasTypeDefinition)
      Reference = ns=1;i=5015 (ReferenceType=HasComponent, IsForward=false)
  UAVariable (DataType=Float, ParentNodeId=ns=1;i=5015, NodeId=ns=1;i=6043, BrowseName=1:Temperature)
    DisplayName = Temperature
    Description = Actual room temperature
    References:
      Reference = i=63 (ReferenceType=HasTypeDefinition)
      Reference = ns=1;i=5015 (ReferenceType=HasComponent, IsForward=false)
  UAVariable (DataType=String, ParentNodeId=ns=1;i=5013, NodeId=ns=1;i=6095, BrowseName=1:Name)
    DisplayName = Name
    Description = Name of the instance
    References:
      Reference = i=63 (ReferenceType=HasTypeDefinition)
      Reference = ns=1;i=5013 (ReferenceType=HasComponent, IsForward=false)
  UAObject (ParentNodeId=ns=1;i=5013, NodeId=ns=1;i=5016, BrowseName=1:Set)
    DisplayName = Set
    Description = Set values
    References:
      Reference = ns=1;i=1004 (ReferenceType=HasTypeDefinition)
      Reference = ns=1;i=6044 (ReferenceType=HasComponent)
      Reference = ns=1;i=5013 (ReferenceType=HasComponent, IsForward=false)
      Reference = ns=1;i=6045 (ReferenceType=HasComponent)
  UAVariable (DataType=Byte, ParentNodeId=ns=1;i=5016, NodeId=ns=1;i=6044, BrowseName=1:FanLevel, AccessLevel=3)
    DisplayName = FanLevel
    Description = The set fan level for operation mode manual
    References:
      Reference = i=63 (ReferenceType=HasTypeDefinition)
      Reference = ns=1;i=5016 (ReferenceType=HasComponent, IsForward=false)
  UAVariable (DataType=Float, ParentNodeId=ns=1;i=5016, NodeId=ns=1;i=6045, BrowseName=1:Temperature, AccessLevel=3)
    DisplayName = Temperature
    Description = The set temperature for operation mode automatic
    References:
      Reference = i=63 (ReferenceType=HasTypeDefinition)
      Reference = ns=1;i=5016 (ReferenceType=HasComponent, IsForward=false)
  UAMethod (ParentNodeId=ns=1;i=5013, NodeId=ns=1;i=7005, BrowseName=1:SetOperationMode, MethodDeclarationId=ns=1;i=7001)
    DisplayName = SetOperationMode
    Description = Set the operation mode of the air condition to Off, Manual or Auto
    References:
      Reference = ns=1;i=6060 (ReferenceType=HasProperty)
      Reference = ns=1;i=6067 (ReferenceType=HasProperty)
      Reference = ns=1;i=5013 (ReferenceType=HasComponent, IsForward=false)
  UAVariable (DataType=Argument, ParentNodeId=ns=1;i=7005, ValueRank=1, NodeId=ns=1;i=6060, ArrayDimensions=1, BrowseName=InputArguments)
    DisplayName = InputArguments
    References:
      Reference = i=68 (ReferenceType=HasTypeDefinition)
      Reference = ns=1;i=7005 (ReferenceType=HasProperty, IsForward=false)
    Value:
      ListOfExtensionObject:
        ExtensionObject:
          TypeId:
            Identifier = i=297
          Body:
            Argument:
              Name = OperationMode
              DataType:
                Identifier = ns=1;i=3002
              ValueRank = -1
              ArrayDimensions
              Description:
                Text = OperationMode (Off, Manual or Automatic)
  UAVariable (DataType=Argument, ParentNodeId=ns=1;i=7005, ValueRank=1, NodeId=ns=1;i=6067, ArrayDimensions=1, BrowseName=OutputArguments)
    DisplayName = OutputArguments
    References:
      Reference = i=68 (ReferenceType=HasTypeDefinition)
      Reference = ns=1;i=7005 (ReferenceType=HasProperty, IsForward=false)
    Value:
      ListOfExtensionObject:
        ExtensionObject:
          TypeId:
            Identifier = i=297
          Body:
            Argument:
              Name = Status
              DataType:
                Identifier = ns=1;i=3003
              ValueRank = -1
              ArrayDimensions
              Description:
                Text = Status of the method
  UAObject (ParentNodeId=ns=1;i=5014, EventNotifier=1, NodeId=ns=1;i=5017, BrowseName=1:Corridor)
    DisplayName = Corridor
    Description = Corridor air condition
    References:
      Reference = ns=1;i=5018 (ReferenceType=HasComponent)
      Reference = ns=1;i=1002 (ReferenceType=GeneratesEvent)
      Reference = ns=1;i=1005 (ReferenceType=HasTypeDefinition)
      Reference = ns=1;i=5014 (ReferenceType=HasComponent, IsForward=false)
      Reference = ns=1;i=6096 (ReferenceType=HasComponent)
      Reference = ns=1;i=5019 (ReferenceType=HasComponent)
      Reference = ns=1;i=7006 (ReferenceType=HasComponent)
      Reference = i=2253 (ReferenceType=HasNotifier, IsForward=false)
  UAObject (ParentNodeId=ns=1;i=5017, NodeId=ns=1;i=5018, BrowseName=1:Act)
    DisplayName = Act
    Description = Actual values
    References:
      Reference = ns=1;i=5017 (ReferenceType=HasComponent, IsForward=false)
      Reference = ns=1;i=1003 (ReferenceType=HasTypeDefinition)
      Reference = ns=1;i=6046 (ReferenceType=HasComponent)
      Reference = ns=1;i=6047 (ReferenceType=HasComponent)
      Reference = ns=1;i=6048 (ReferenceType=HasComponent)
  UAVariable (DataType=Byte, ParentNodeId=ns=1;i=5018, NodeId=ns=1;i=6046, BrowseName=1:FanLevel)
    DisplayName = FanLevel
    Description = Actual level of the fan
    References:
      Reference = i=63 (ReferenceType=HasTypeDefinition)
      Reference = ns=1;i=5018 (ReferenceType=HasComponent, IsForward=false)
  UAVariable (DataType=Int32, ParentNodeId=ns=1;i=5018, NodeId=ns=1;i=6047, BrowseName=1:OperationMode)
    DisplayName = OperationMode
    Description = Actual operation mode of the air condtition: Off, Manual or Auto
    References:
      Reference = i=63 (ReferenceType=HasTypeDefinition)
      Reference = ns=1;i=5018 (ReferenceType=HasComponent, IsForward=false)
  UAVariable (DataType=Float, ParentNodeId=ns=1;i=5018, NodeId=ns=1;i=6048, BrowseName=1:Temperature)
    DisplayName = Temperature
    Description = Actual room temperature
    References:
      Reference = i=63 (ReferenceType=HasTypeDefinition)
      Reference = ns=1;i=5018 (ReferenceType=HasComponent, IsForward=false)
  UAVariable (DataType=String, ParentNodeId=ns=1;i=5017, NodeId=ns=1;i=6096, BrowseName=1:Name)
    DisplayName = Name
    Description = Name of the instance
    References:
      Reference = i=63 (ReferenceType=HasTypeDefinition)
      Reference = ns=1;i=5017 (ReferenceType=HasComponent, IsForward=false)
  UAObject (ParentNodeId=ns=1;i=5017, NodeId=ns=1;i=5019, BrowseName=1:Set)
    DisplayName = Set
    Description = Set values
    References:
      Reference = ns=1;i=1004 (ReferenceType=HasTypeDefinition)
      Reference = ns=1;i=6049 (ReferenceType=HasComponent)
      Reference = ns=1;i=5017 (ReferenceType=HasComponent, IsForward=false)
      Reference = ns=1;i=6050 (ReferenceType=HasComponent)
  UAVariable (DataType=Byte, ParentNodeId=ns=1;i=5019, NodeId=ns=1;i=6049, BrowseName=1:FanLevel, AccessLevel=3)
    DisplayName = FanLevel
    Description = The set fan level for operation mode manual
    References:
      Reference = i=63 (ReferenceType=HasTypeDefinition)
      Reference = ns=1;i=5019 (ReferenceType=HasComponent, IsForward=false)
  UAVariable (DataType=Float, ParentNodeId=ns=1;i=5019, NodeId=ns=1;i=6050, BrowseName=1:Temperature, AccessLevel=3)
    DisplayName = Temperature
    Description = The set temperature for operation mode automatic
    References:
      Reference = i=63 (ReferenceType=HasTypeDefinition)
      Reference = ns=1;i=5019 (ReferenceType=HasComponent, IsForward=false)
  UAMethod (ParentNodeId=ns=1;i=5017, NodeId=ns=1;i=7006, BrowseName=1:SetOperationMode, MethodDeclarationId=ns=1;i=7001)
    DisplayName = SetOperationMode
    Description = Set the operation mode of the air condition to Off, Manual or Auto
    References:
      Reference = ns=1;i=6061 (ReferenceType=HasProperty)
      Reference = ns=1;i=6068 (ReferenceType=HasProperty)
      Reference = ns=1;i=5017 (ReferenceType=HasComponent, IsForward=false)
  UAVariable (DataType=Argument, ParentNodeId=ns=1;i=7006, ValueRank=1, NodeId=ns=1;i=6061, ArrayDimensions=1, BrowseName=InputArguments)
    DisplayName = InputArguments
    References:
      Reference = i=68 (ReferenceType=HasTypeDefinition)
      Reference = ns=1;i=7006 (ReferenceType=HasProperty, IsForward=false)
    Value:
      ListOfExtensionObject:
        ExtensionObject:
          TypeId:
            Identifier = i=297
          Body:
            Argument:
              Name = OperationMode
              DataType:
                Identifier = ns=1;i=3002
              ValueRank = -1
              ArrayDimensions
              Description:
                Text = OperationMode (Off, Manual or Automatic)
  UAVariable (DataType=Argument, ParentNodeId=ns=1;i=7006, ValueRank=1, NodeId=ns=1;i=6068, ArrayDimensions=1, BrowseName=OutputArguments)
    DisplayName = OutputArguments
    References:
      Reference = i=68 (ReferenceType=HasTypeDefinition)
      Reference = ns=1;i=7006 (ReferenceType=HasProperty, IsForward=false)
    Value:
      ListOfExtensionObject:
        ExtensionObject:
          TypeId:
            Identifier = i=297
          Body:
            Argument:
              Name = Status
              DataType:
                Identifier = ns=1;i=3003
              ValueRank = -1
              ArrayDimensions
              Description:
                Text = Status of the method
  UAObject (ParentNodeId=ns=1;i=5014, EventNotifier=1, NodeId=ns=1;i=5020, BrowseName=1:LivingRoom)
    DisplayName = LivingRoom
    Description = Living room air condition
    References:
      Reference = ns=1;i=5021 (ReferenceType=HasComponent)
      Reference = ns=1;i=1002 (ReferenceType=GeneratesEvent)
      Reference = ns=1;i=1005 (ReferenceType=HasTypeDefinition)
      Reference = ns=1;i=5014 (ReferenceType=HasComponent, IsForward=false)
      Reference = ns=1;i=6097 (ReferenceType=HasComponent)
      Reference = ns=1;i=5022 (ReferenceType=HasComponent)
      Reference = ns=1;i=7007 (ReferenceType=HasComponent)
      Reference = i=2253 (ReferenceType=HasNotifier, IsForward=false)
  UAObject (ParentNodeId=ns=1;i=5020, NodeId=ns=1;i=5021, BrowseName=1:Act)
    DisplayName = Act
    Description = Actual values
    References:
      Reference = ns=1;i=5020 (ReferenceType=HasComponent, IsForward=false)
      Reference = ns=1;i=1003 (ReferenceType=HasTypeDefinition)
      Reference = ns=1;i=6051 (ReferenceType=HasComponent)
      Reference = ns=1;i=6052 (ReferenceType=HasComponent)
      Reference = ns=1;i=6053 (ReferenceType=HasComponent)
  UAVariable (DataType=Byte, ParentNodeId=ns=1;i=5021, NodeId=ns=1;i=6051, BrowseName=1:FanLevel)
    DisplayName = FanLevel
    Description = Actual level of the fan
    References:
      Reference = i=63 (ReferenceType=HasTypeDefinition)
      Reference = ns=1;i=5021 (ReferenceType=HasComponent, IsForward=false)
  UAVariable (DataType=Int32, ParentNodeId=ns=1;i=5021, NodeId=ns=1;i=6052, BrowseName=1:OperationMode)
    DisplayName = OperationMode
    Description = Actual operation mode of the air condtition: Off, Manual or Auto
    References:
      Reference = i=63 (ReferenceType=HasTypeDefinition)
      Reference = ns=1;i=5021 (ReferenceType=HasComponent, IsForward=false)
  UAVariable (DataType=Float, ParentNodeId=ns=1;i=5021, NodeId=ns=1;i=6053, BrowseName=1:Temperature)
    DisplayName = Temperature
    Description = Actual room temperature
    References:
      Reference = i=63 (ReferenceType=HasTypeDefinition)
      Reference = ns=1;i=5021 (ReferenceType=HasComponent, IsForward=false)
  UAVariable (DataType=String, ParentNodeId=ns=1;i=5020, NodeId=ns=1;i=6097, BrowseName=1:Name)
    DisplayName = Name
    Description = Name of the instance
    References:
      Reference = i=63 (ReferenceType=HasTypeDefinition)
      Reference = ns=1;i=5020 (ReferenceType=HasComponent, IsForward=false)
  UAObject (ParentNodeId=ns=1;i=5020, NodeId=ns=1;i=5022, BrowseName=1:Set)
    DisplayName = Set
    Description = Set values
    References:
      Reference = ns=1;i=1004 (ReferenceType=HasTypeDefinition)
      Reference = ns=1;i=6054 (ReferenceType=HasComponent)
      Reference = ns=1;i=5020 (ReferenceType=HasComponent, IsForward=false)
      Reference = ns=1;i=6055 (ReferenceType=HasComponent)
  UAVariable (DataType=Byte, ParentNodeId=ns=1;i=5022, NodeId=ns=1;i=6054, BrowseName=1:FanLevel, AccessLevel=3)
    DisplayName = FanLevel
    Description = The set fan level for operation mode manual
    References:
      Reference = i=63 (ReferenceType=HasTypeDefinition)
      Reference = ns=1;i=5022 (ReferenceType=HasComponent, IsForward=false)
  UAVariable (DataType=Float, ParentNodeId=ns=1;i=5022, NodeId=ns=1;i=6055, BrowseName=1:Temperature, AccessLevel=3)
    DisplayName = Temperature
    Description = The set temperature for operation mode automatic
    References:
      Reference = i=63 (ReferenceType=HasTypeDefinition)
      Reference = ns=1;i=5022 (ReferenceType=HasComponent, IsForward=false)
  UAMethod (ParentNodeId=ns=1;i=5020, NodeId=ns=1;i=7007, BrowseName=1:SetOperationMode, MethodDeclarationId=ns=1;i=7001)
    DisplayName = SetOperationMode
    Description = Set the operation mode of the air condition to Off, Manual or Auto
    References:
      Reference = ns=1;i=6062 (ReferenceType=HasProperty)
      Reference = ns=1;i=6069 (ReferenceType=HasProperty)
      Reference = ns=1;i=5020 (ReferenceType=HasComponent, IsForward=false)
  UAVariable (DataType=Argument, ParentNodeId=ns=1;i=7007, ValueRank=1, NodeId=ns=1;i=6062, ArrayDimensions=1, BrowseName=InputArguments)
    DisplayName = InputArguments
    References:
      Reference = i=68 (ReferenceType=HasTypeDefinition)
      Reference = ns=1;i=7007 (ReferenceType=HasProperty, IsForward=false)
    Value:
      ListOfExtensionObject:
        ExtensionObject:
          TypeId:
            Identifier = i=297
          Body:
            Argument:
              Name = OperationMode
              DataType:
                Identifier = ns=1;i=3002
              ValueRank = -1
              ArrayDimensions
              Description:
                Text = OperationMode (Off, Manual or Automatic)
  UAVariable (DataType=Argument, ParentNodeId=ns=1;i=7007, ValueRank=1, NodeId=ns=1;i=6069, ArrayDimensions=1, BrowseName=OutputArguments)
    DisplayName = OutputArguments
    References:
      Reference = i=68 (ReferenceType=HasTypeDefinition)
      Reference = ns=1;i=7007 (ReferenceType=HasProperty, IsForward=false)
    Value:
      ListOfExtensionObject:
        ExtensionObject:
          TypeId:
            Identifier = i=297
          Body:
            Argument:
              Name = Status
              DataType:
                Identifier = ns=1;i=3003
              ValueRank = -1
              ArrayDimensions
              Description:
                Text = Status of the method
  UAObject (NodeId=ns=1;i=5024, BrowseName=1:ST)
    DisplayName = ST
    Description = Root of all air conditions in variant of StructuredText
    References:
      Reference = ns=1;i=1006 (ReferenceType=HasTypeDefinition)
      Reference = ns=1;i=5023 (ReferenceType=HasComponent)
      Reference = ns=1;i=5027 (ReferenceType=HasComponent)
      Reference = ns=1;i=5030 (ReferenceType=HasComponent)
      Reference = ns=1;i=5033 (ReferenceType=Organizes, IsForward=false)
  UAObject (ParentNodeId=ns=1;i=5024, EventNotifier=1, NodeId=ns=1;i=5023, BrowseName=1:BedRoom)
    DisplayName = BedRoom
    Description = Bed room air condition
    References:
      Reference = ns=1;i=5025 (ReferenceType=HasComponent)
      Reference = ns=1;i=1002 (ReferenceType=GeneratesEvent)
      Reference = ns=1;i=1005 (ReferenceType=HasTypeDefinition)
      Reference = ns=1;i=6098 (ReferenceType=HasComponent)
      Reference = ns=1;i=5026 (ReferenceType=HasComponent)
      Reference = ns=1;i=7008 (ReferenceType=HasComponent)
      Reference = i=2253 (ReferenceType=HasNotifier, IsForward=false)
      Reference = ns=1;i=5024 (ReferenceType=HasComponent, IsForward=false)
  UAObject (ParentNodeId=ns=1;i=5023, NodeId=ns=1;i=5025, BrowseName=1:Act)
    DisplayName = Act
    Description = Actual values
    References:
      Reference = ns=1;i=5023 (ReferenceType=HasComponent, IsForward=false)
      Reference = ns=1;i=1003 (ReferenceType=HasTypeDefinition)
      Reference = ns=1;i=6070 (ReferenceType=HasComponent)
      Reference = ns=1;i=6071 (ReferenceType=HasComponent)
      Reference = ns=1;i=6072 (ReferenceType=HasComponent)
  UAVariable (DataType=Byte, ParentNodeId=ns=1;i=5025, NodeId=ns=1;i=6070, BrowseName=1:FanLevel)
    DisplayName = FanLevel
    Description = Actual level of the fan
    References:
      Reference = i=63 (ReferenceType=HasTypeDefinition)
      Reference = ns=1;i=5025 (ReferenceType=HasComponent, IsForward=false)
  UAVariable (DataType=Int32, ParentNodeId=ns=1;i=5025, NodeId=ns=1;i=6071, BrowseName=1:OperationMode)
    DisplayName = OperationMode
    Description = Actual operation mode of the air condtition: Off, Manual or Auto
    References:
      Reference = i=63 (ReferenceType=HasTypeDefinition)
      Reference = ns=1;i=5025 (ReferenceType=HasComponent, IsForward=false)
  UAVariable (DataType=Float, ParentNodeId=ns=1;i=5025, NodeId=ns=1;i=6072, BrowseName=1:Temperature)
    DisplayName = Temperature
    Description = Actual room temperature
    References:
      Reference = i=63 (ReferenceType=HasTypeDefinition)
      Reference = ns=1;i=5025 (ReferenceType=HasComponent, IsForward=false)
  UAVariable (DataType=String, ParentNodeId=ns=1;i=5023, NodeId=ns=1;i=6098, BrowseName=1:Name)
    DisplayName = Name
    Description = Name of the instance
    References:
      Reference = i=63 (ReferenceType=HasTypeDefinition)
      Reference = ns=1;i=5023 (ReferenceType=HasComponent, IsForward=false)
  UAObject (ParentNodeId=ns=1;i=5023, NodeId=ns=1;i=5026, BrowseName=1:Set)
    DisplayName = Set
    Description = Set values
    References:
      Reference = ns=1;i=1004 (ReferenceType=HasTypeDefinition)
      Reference = ns=1;i=6073 (ReferenceType=HasComponent)
      Reference = ns=1;i=5023 (ReferenceType=HasComponent, IsForward=false)
      Reference = ns=1;i=6074 (ReferenceType=HasComponent)
  UAVariable (DataType=Byte, ParentNodeId=ns=1;i=5026, NodeId=ns=1;i=6073, BrowseName=1:FanLevel, AccessLevel=3)
    DisplayName = FanLevel
    Description = The set fan level for operation mode manual
    References:
      Reference = i=63 (ReferenceType=HasTypeDefinition)
      Reference = ns=1;i=5026 (ReferenceType=HasComponent, IsForward=false)
  UAVariable (DataType=Float, ParentNodeId=ns=1;i=5026, NodeId=ns=1;i=6074, BrowseName=1:Temperature, AccessLevel=3)
    DisplayName = Temperature
    Description = The set temperature for operation mode automatic
    References:
      Reference = i=63 (ReferenceType=HasTypeDefinition)
      Reference = ns=1;i=5026 (ReferenceType=HasComponent, IsForward=false)
  UAMethod (ParentNodeId=ns=1;i=5023, NodeId=ns=1;i=7008, BrowseName=1:SetOperationMode, MethodDeclarationId=ns=1;i=7001)
    DisplayName = SetOperationMode
    Description = Set the operation mode of the air condition to Off, Manual or Auto
    References:
      Reference = ns=1;i=6075 (ReferenceType=HasProperty)
      Reference = ns=1;i=6076 (ReferenceType=HasProperty)
      Reference = ns=1;i=5023 (ReferenceType=HasComponent, IsForward=false)
  UAVariable (DataType=Argument, ParentNodeId=ns=1;i=7008, ValueRank=1, NodeId=ns=1;i=6075, ArrayDimensions=1, BrowseName=InputArguments)
    DisplayName = InputArguments
    References:
      Reference = i=68 (ReferenceType=HasTypeDefinition)
      Reference = ns=1;i=7008 (ReferenceType=HasProperty, IsForward=false)
    Value:
      ListOfExtensionObject:
        ExtensionObject:
          TypeId:
            Identifier = i=297
          Body:
            Argument:
              Name = OperationMode
              DataType:
                Identifier = ns=1;i=3002
              ValueRank = -1
              ArrayDimensions
              Description:
                Text = OperationMode (Off, Manual or Automatic)
  UAVariable (DataType=Argument, ParentNodeId=ns=1;i=7008, ValueRank=1, NodeId=ns=1;i=6076, ArrayDimensions=1, BrowseName=OutputArguments)
    DisplayName = OutputArguments
    References:
      Reference = i=68 (ReferenceType=HasTypeDefinition)
      Reference = ns=1;i=7008 (ReferenceType=HasProperty, IsForward=false)
    Value:
      ListOfExtensionObject:
        ExtensionObject:
          TypeId:
            Identifier = i=297
          Body:
            Argument:
              Name = Status
              DataType:
                Identifier = ns=1;i=3003
              ValueRank = -1
              ArrayDimensions
              Description:
                Text = Status of the method
  UAObject (ParentNodeId=ns=1;i=5024, EventNotifier=1, NodeId=ns=1;i=5027, BrowseName=1:Corridor)
    DisplayName = Corridor
    Description = Corridor air condition
    References:
      Reference = ns=1;i=5028 (ReferenceType=HasComponent)
      Reference = ns=1;i=1002 (ReferenceType=GeneratesEvent)
      Reference = ns=1;i=1005 (ReferenceType=HasTypeDefinition)
      Reference = ns=1;i=5024 (ReferenceType=HasComponent, IsForward=false)
      Reference = ns=1;i=6099 (ReferenceType=HasComponent)
      Reference = ns=1;i=5029 (ReferenceType=HasComponent)
      Reference = ns=1;i=7009 (ReferenceType=HasComponent)
      Reference = i=2253 (ReferenceType=HasNotifier, IsForward=false)
  UAObject (ParentNodeId=ns=1;i=5027, NodeId=ns=1;i=5028, BrowseName=1:Act)
    DisplayName = Act
    Description = Actual values
    References:
      Reference = ns=1;i=5027 (ReferenceType=HasComponent, IsForward=false)
      Reference = ns=1;i=1003 (ReferenceType=HasTypeDefinition)
      Reference = ns=1;i=6077 (ReferenceType=HasComponent)
      Reference = ns=1;i=6078 (ReferenceType=HasComponent)
      Reference = ns=1;i=6079 (ReferenceType=HasComponent)
  UAVariable (DataType=Byte, ParentNodeId=ns=1;i=5028, NodeId=ns=1;i=6077, BrowseName=1:FanLevel)
    DisplayName = FanLevel
    Description = Actual level of the fan
    References:
      Reference = i=63 (ReferenceType=HasTypeDefinition)
      Reference = ns=1;i=5028 (ReferenceType=HasComponent, IsForward=false)
  UAVariable (DataType=Int32, ParentNodeId=ns=1;i=5028, NodeId=ns=1;i=6078, BrowseName=1:OperationMode)
    DisplayName = OperationMode
    Description = Actual operation mode of the air condtition: Off, Manual or Auto
    References:
      Reference = i=63 (ReferenceType=HasTypeDefinition)
      Reference = ns=1;i=5028 (ReferenceType=HasComponent, IsForward=false)
  UAVariable (DataType=Float, ParentNodeId=ns=1;i=5028, NodeId=ns=1;i=6079, BrowseName=1:Temperature)
    DisplayName = Temperature
    Description = Actual room temperature
    References:
      Reference = i=63 (ReferenceType=HasTypeDefinition)
      Reference = ns=1;i=5028 (ReferenceType=HasComponent, IsForward=false)
  UAVariable (DataType=String, ParentNodeId=ns=1;i=5027, NodeId=ns=1;i=6099, BrowseName=1:Name)
    DisplayName = Name
    Description = Name of the instance
    References:
      Reference = i=63 (ReferenceType=HasTypeDefinition)
      Reference = ns=1;i=5027 (ReferenceType=HasComponent, IsForward=false)
  UAObject (ParentNodeId=ns=1;i=5027, NodeId=ns=1;i=5029, BrowseName=1:Set)
    DisplayName = Set
    Description = Set values
    References:
      Reference = ns=1;i=1004 (ReferenceType=HasTypeDefinition)
      Reference = ns=1;i=6080 (ReferenceType=HasComponent)
      Reference = ns=1;i=5027 (ReferenceType=HasComponent, IsForward=false)
      Reference = ns=1;i=6081 (ReferenceType=HasComponent)
  UAVariable (DataType=Byte, ParentNodeId=ns=1;i=5029, NodeId=ns=1;i=6080, BrowseName=1:FanLevel, AccessLevel=3)
    DisplayName = FanLevel
    Description = The set fan level for operation mode manual
    References:
      Reference = i=63 (ReferenceType=HasTypeDefinition)
      Reference = ns=1;i=5029 (ReferenceType=HasComponent, IsForward=false)
  UAVariable (DataType=Float, ParentNodeId=ns=1;i=5029, NodeId=ns=1;i=6081, BrowseName=1:Temperature, AccessLevel=3)
    DisplayName = Temperature
    Description = The set temperature for operation mode automatic
    References:
      Reference = i=63 (ReferenceType=HasTypeDefinition)
      Reference = ns=1;i=5029 (ReferenceType=HasComponent, IsForward=false)
  UAMethod (ParentNodeId=ns=1;i=5027, NodeId=ns=1;i=7009, BrowseName=1:SetOperationMode, MethodDeclarationId=ns=1;i=7001)
    DisplayName = SetOperationMode
    Description = Set the operation mode of the air condition to Off, Manual or Auto
    References:
      Reference = ns=1;i=6082 (ReferenceType=HasProperty)
      Reference = ns=1;i=6083 (ReferenceType=HasProperty)
      Reference = ns=1;i=5027 (ReferenceType=HasComponent, IsForward=false)
  UAVariable (DataType=Argument, ParentNodeId=ns=1;i=7009, ValueRank=1, NodeId=ns=1;i=6082, ArrayDimensions=1, BrowseName=InputArguments)
    DisplayName = InputArguments
    References:
      Reference = i=68 (ReferenceType=HasTypeDefinition)
      Reference = ns=1;i=7009 (ReferenceType=HasProperty, IsForward=false)
    Value:
      ListOfExtensionObject:
        ExtensionObject:
          TypeId:
            Identifier = i=297
          Body:
            Argument:
              Name = OperationMode
              DataType:
                Identifier = ns=1;i=3002
              ValueRank = -1
              ArrayDimensions
              Description:
                Text = OperationMode (Off, Manual or Automatic)
  UAVariable (DataType=Argument, ParentNodeId=ns=1;i=7009, ValueRank=1, NodeId=ns=1;i=6083, ArrayDimensions=1, BrowseName=OutputArguments)
    DisplayName = OutputArguments
    References:
      Reference = i=68 (ReferenceType=HasTypeDefinition)
      Reference = ns=1;i=7009 (ReferenceType=HasProperty, IsForward=false)
    Value:
      ListOfExtensionObject:
        ExtensionObject:
          TypeId:
            Identifier = i=297
          Body:
            Argument:
              Name = Status
              DataType:
                Identifier = ns=1;i=3003
              ValueRank = -1
              ArrayDimensions
              Description:
                Text = Status of the method
  UAObject (ParentNodeId=ns=1;i=5024, EventNotifier=1, NodeId=ns=1;i=5030, BrowseName=1:LivingRoom)
    DisplayName = LivingRoom
    Description = Living room air condition
    References:
      Reference = ns=1;i=5031 (ReferenceType=HasComponent)
      Reference = ns=1;i=1002 (ReferenceType=GeneratesEvent)
      Reference = ns=1;i=1005 (ReferenceType=HasTypeDefinition)
      Reference = ns=1;i=5024 (ReferenceType=HasComponent, IsForward=false)
      Reference = ns=1;i=6100 (ReferenceType=HasComponent)
      Reference = ns=1;i=5032 (ReferenceType=HasComponent)
      Reference = ns=1;i=7010 (ReferenceType=HasComponent)
      Reference = i=2253 (ReferenceType=HasNotifier, IsForward=false)
  UAObject (ParentNodeId=ns=1;i=5030, NodeId=ns=1;i=5031, BrowseName=1:Act)
    DisplayName = Act
    Description = Actual values
    References:
      Reference = ns=1;i=5030 (ReferenceType=HasComponent, IsForward=false)
      Reference = ns=1;i=1003 (ReferenceType=HasTypeDefinition)
      Reference = ns=1;i=6084 (ReferenceType=HasComponent)
      Reference = ns=1;i=6085 (ReferenceType=HasComponent)
      Reference = ns=1;i=6086 (ReferenceType=HasComponent)
  UAVariable (DataType=Byte, ParentNodeId=ns=1;i=5031, NodeId=ns=1;i=6084, BrowseName=1:FanLevel)
    DisplayName = FanLevel
    Description = Actual level of the fan
    References:
      Reference = i=63 (ReferenceType=HasTypeDefinition)
      Reference = ns=1;i=5031 (ReferenceType=HasComponent, IsForward=false)
  UAVariable (DataType=Int32, ParentNodeId=ns=1;i=5031, NodeId=ns=1;i=6085, BrowseName=1:OperationMode)
    DisplayName = OperationMode
    Description = Actual operation mode of the air condtition: Off, Manual or Auto
    References:
      Reference = i=63 (ReferenceType=HasTypeDefinition)
      Reference = ns=1;i=5031 (ReferenceType=HasComponent, IsForward=false)
  UAVariable (DataType=Float, ParentNodeId=ns=1;i=5031, NodeId=ns=1;i=6086, BrowseName=1:Temperature)
    DisplayName = Temperature
    Description = Actual room temperature
    References:
      Reference = i=63 (ReferenceType=HasTypeDefinition)
      Reference = ns=1;i=5031 (ReferenceType=HasComponent, IsForward=false)
  UAVariable (DataType=String, ParentNodeId=ns=1;i=5030, NodeId=ns=1;i=6100, BrowseName=1:Name)
    DisplayName = Name
    Description = Name of the instance
    References:
      Reference = i=63 (ReferenceType=HasTypeDefinition)
      Reference = ns=1;i=5030 (ReferenceType=HasComponent, IsForward=false)
  UAObject (ParentNodeId=ns=1;i=5030, NodeId=ns=1;i=5032, BrowseName=1:Set)
    DisplayName = Set
    Description = Set values
    References:
      Reference = ns=1;i=1004 (ReferenceType=HasTypeDefinition)
      Reference = ns=1;i=6087 (ReferenceType=HasComponent)
      Reference = ns=1;i=5030 (ReferenceType=HasComponent, IsForward=false)
      Reference = ns=1;i=6088 (ReferenceType=HasComponent)
  UAVariable (DataType=Byte, ParentNodeId=ns=1;i=5032, NodeId=ns=1;i=6087, BrowseName=1:FanLevel, AccessLevel=3)
    DisplayName = FanLevel
    Description = The set fan level for operation mode manual
    References:
      Reference = i=63 (ReferenceType=HasTypeDefinition)
      Reference = ns=1;i=5032 (ReferenceType=HasComponent, IsForward=false)
  UAVariable (DataType=Float, ParentNodeId=ns=1;i=5032, NodeId=ns=1;i=6088, BrowseName=1:Temperature, AccessLevel=3)
    DisplayName = Temperature
    Description = The set temperature for operation mode automatic
    References:
      Reference = i=63 (ReferenceType=HasTypeDefinition)
      Reference = ns=1;i=5032 (ReferenceType=HasComponent, IsForward=false)
  UAMethod (ParentNodeId=ns=1;i=5030, NodeId=ns=1;i=7010, BrowseName=1:SetOperationMode, MethodDeclarationId=ns=1;i=7001)
    DisplayName = SetOperationMode
    Description = Set the operation mode of the air condition to Off, Manual or Auto
    References:
      Reference = ns=1;i=6089 (ReferenceType=HasProperty)
      Reference = ns=1;i=6090 (ReferenceType=HasProperty)
      Reference = ns=1;i=5030 (ReferenceType=HasComponent, IsForward=false)
  UAVariable (DataType=Argument, ParentNodeId=ns=1;i=7010, ValueRank=1, NodeId=ns=1;i=6089, ArrayDimensions=1, BrowseName=InputArguments)
    DisplayName = InputArguments
    References:
      Reference = i=68 (ReferenceType=HasTypeDefinition)
      Reference = ns=1;i=7010 (ReferenceType=HasProperty, IsForward=false)
    Value:
      ListOfExtensionObject:
        ExtensionObject:
          TypeId:
            Identifier = i=297
          Body:
            Argument:
              Name = OperationMode
              DataType:
                Identifier = ns=1;i=3002
              ValueRank = -1
              ArrayDimensions
              Description:
                Text = OperationMode (Off, Manual or Automatic)
  UAVariable (DataType=Argument, ParentNodeId=ns=1;i=7010, ValueRank=1, NodeId=ns=1;i=6090, ArrayDimensions=1, BrowseName=OutputArguments)
    DisplayName = OutputArguments
    References:
      Reference = i=68 (ReferenceType=HasTypeDefinition)
      Reference = ns=1;i=7010 (ReferenceType=HasProperty, IsForward=false)
    Value:
      ListOfExtensionObject:
        ExtensionObject:
          TypeId:
            Identifier = i=297
          Body:
            Argument:
              Name = Status
              DataType:
                Identifier = ns=1;i=3003
              ValueRank = -1
              ArrayDimensions
              Description:
                Text = Status of the method
  UAObject (SymbolicName=http___br_automation_com_AirCondModel_, NodeId=ns=1;i=5001, BrowseName=1:http://br-automation.com/AirCondModel/)
    DisplayName = http://br-automation.com/AirCondModel/
    Description = Provides the metadata for a namespace used by the server.
    References:
      Reference = ns=1;i=6001 (ReferenceType=HasProperty)
      Reference = i=11616 (ReferenceType=HasTypeDefinition)
      Reference = i=11715 (ReferenceType=HasComponent, IsForward=false)
      Reference = ns=1;i=6002 (ReferenceType=HasProperty)
      Reference = ns=1;i=6003 (ReferenceType=HasProperty)
      Reference = ns=1;i=6004 (ReferenceType=HasProperty)
      Reference = ns=1;i=6005 (ReferenceType=HasProperty)
      Reference = ns=1;i=6006 (ReferenceType=HasProperty)
      Reference = ns=1;i=6007 (ReferenceType=HasProperty)
  UAVariable (DataType=Boolean, ParentNodeId=ns=1;i=5001, NodeId=ns=1;i=6001, BrowseName=IsNamespaceSubset)
    DisplayName = IsNamespaceSubset
    Description = If TRUE then the server only supports a subset of the namespace.
    References:
      Reference = ns=1;i=5001 (ReferenceType=HasProperty, IsForward=false)
      Reference = i=68 (ReferenceType=HasTypeDefinition)
    Value:
      Boolean = false
  UAVariable (DataType=DateTime, ParentNodeId=ns=1;i=5001, NodeId=ns=1;i=6002, BrowseName=NamespacePublicationDate)
    DisplayName = NamespacePublicationDate
    Description = The publication date for the namespace.
    References:
      Reference = ns=1;i=5001 (ReferenceType=HasProperty, IsForward=false)
      Reference = i=68 (ReferenceType=HasTypeDefinition)
    Value:
      DateTime = 2020-07-13T13:29:09Z
  UAVariable (DataType=String, ParentNodeId=ns=1;i=5001, NodeId=ns=1;i=6003, BrowseName=NamespaceUri)
    DisplayName = NamespaceUri
    Description = The URI of the namespace.
    References:
      Reference = ns=1;i=5001 (ReferenceType=HasProperty, IsForward=false)
      Reference = i=68 (ReferenceType=HasTypeDefinition)
    Value:
      String = http://br-automation.com/AirCondModel/
  UAVariable (DataType=String, ParentNodeId=ns=1;i=5001, NodeId=ns=1;i=6004, BrowseName=NamespaceVersion)
    DisplayName = NamespaceVersion
    Description = The human readable string representing version of the namespace.
    References:
      Reference = ns=1;i=5001 (ReferenceType=HasProperty, IsForward=false)
      Reference = i=68 (ReferenceType=HasTypeDefinition)
    Value:
      String = 1.0.0
  UAVariable (DataType=IdType, ParentNodeId=ns=1;i=5001, ValueRank=1, NodeId=ns=1;i=6005, BrowseName=StaticNodeIdTypes)
    DisplayName = StaticNodeIdTypes
    Description = A list of IdTypes for nodes which are the same in every server that exposes them.
    References:
      Reference = i=68 (ReferenceType=HasTypeDefinition)
      Reference = ns=1;i=5001 (ReferenceType=HasProperty, IsForward=false)
  UAVariable (DataType=NumericRange, ParentNodeId=ns=1;i=5001, ValueRank=1, NodeId=ns=1;i=6006, BrowseName=StaticNumericNodeIdRange)
    DisplayName = StaticNumericNodeIdRange
    Description = A list of ranges for numeric node ids which are the same in every server that exposes them.
    References:
      Reference = i=68 (ReferenceType=HasTypeDefinition)
      Reference = ns=1;i=5001 (ReferenceType=HasProperty, IsForward=false)
  UAVariable (DataType=String, ParentNodeId=ns=1;i=5001, NodeId=ns=1;i=6007, BrowseName=StaticStringNodeIdPattern)
    DisplayName = StaticStringNodeIdPattern
    Description = A regular expression which matches string node ids are the same in every server that exposes them.
    References:
      Reference = i=68 (ReferenceType=HasTypeDefinition)
      Reference = ns=1;i=5001 (ReferenceType=HasProperty, IsForward=false)
```

### IoMap.iom - X20CP0483/IoMap.iom
```iecst
(********************************************************************
 * COPYRIGHT -- Bernecker + Rainer
 ********************************************************************
 * File: IoMap.iom
 * Author: niedermeierr
 * Created: July 26, 2018
 ********************************************************************
 * IO mapping file
 ********************************************************************)
VAR_CONFIG
	::OpcUaAny:Data.Read.Client.nUsint AT %IB."OpcUa_any".Read_Usint;
	::OpcUaAny:Data.Read.Client.nUint AT %IW."OpcUa_any".Read_Uint;
	::OpcUaAny:Data.Read.Client.nUdint AT %ID."OpcUa_any".Read_Udint;
	::OpcUaAny:Data.Write.Client.nUsint AT %QB."OpcUa_any".Write_Usint;
	::OpcUaAny:Data.Write.Client.nUint AT %QW."OpcUa_any".Write_Uint;
	::OpcUaAny:Data.Write.Client.nUdint AT %QD."OpcUa_any".Write_Udint;
END_VAR
```

## Logical view

Binary libraries used (declarations not repeated): ArCert, ArEventLog, ArPubSubD, ArSsl, AsBrStr, AsBrWStr, AsIecCon, AsOpcUac, AsOpcUas, AsTime, AsUSB, Operator, Runtime, standard, sys_lib, FileIO, DataObj, UnitTest, UtMgr, UtWs
